   "Area03_Messages".W.Msg[#WngIndex + 0] := "A0301_Fermi_P4".Warning.Fermi[1].NotAutReady;
   "Area03_Messages".W.Msg[#WngIndex + 1] := "A0301_Fermi_P4".Warning.Fermi[1].PressureRunning_Timeout;
   "Area03_Messages".W.Msg[#WngIndex + 2] := "A0301_Fermi_P4".Warning.Fermi[1].Rest_MissingExtEnable;
   "Area03_Messages".W.Msg[#WngIndex + 3] := "A0301_Fermi_P4".Warning.Fermi[1].Work_MissingExtEnable;
   "Area03_Messages".W.Msg[#WngIndex + 4] := "A0301_Fermi_P4".Warning.Fermi[1].Missing_Rest_Ls_ON[1];
   "Area03_Messages".W.Msg[#WngIndex + 5] := "A0301_Fermi_P4".Warning.Fermi[1].Missing_Work_Ls_ON[1];
   "Area03_Messages".W.Msg[#WngIndex + 6] := "A0301_Fermi_P4".Warning.Fermi[2].NotAutReady;
   "Area03_Messages".W.Msg[#WngIndex + 7] := "A0301_Fermi_P4".Warning.Fermi[2].PressureRunning_Timeout;
   "Area03_Messages".W.Msg[#WngIndex + 8] := "A0301_Fermi_P4".Warning.Fermi[2].Rest_MissingExtEnable;
   "Area03_Messages".W.Msg[#WngIndex + 9] := "A0301_Fermi_P4".Warning.Fermi[2].Work_MissingExtEnable;
   "Area03_Messages".W.Msg[#WngIndex + 10] := "A0301_Fermi_P4".Warning.Fermi[2].Missing_Rest_Ls_ON[1];
   "Area03_Messages".W.Msg[#WngIndex + 11] := "A0301_Fermi_P4".Warning.Fermi[2].Missing_Work_Ls_ON[1];
   "Area03_Messages".W.Msg[#WngIndex + 12] := "A0301_Fermi_P4".Warning.Fermi[3].NotAutReady;
   "Area03_Messages".W.Msg[#WngIndex + 13] := "A0301_Fermi_P4".Warning.Fermi[3].PressureRunning_Timeout;
   "Area03_Messages".W.Msg[#WngIndex + 14] := "A0301_Fermi_P4".Warning.Fermi[3].Rest_MissingExtEnable;
   "Area03_Messages".W.Msg[#WngIndex + 15] := "A0301_Fermi_P4".Warning.Fermi[3].Work_MissingExtEnable;
   "Area03_Messages".W.Msg[#WngIndex + 16] := "A0301_Fermi_P4".Warning.Fermi[3].Missing_Rest_Ls_ON[1];
   "Area03_Messages".W.Msg[#WngIndex + 17] := "A0301_Fermi_P4".Warning.Fermi[3].Missing_Work_Ls_ON[1];
   "Area03_Messages".W.Msg[#WngIndex + 18] := "A0301_Fermi_P4".Warning.Fermi[4].NotAutReady;
   "Area03_Messages".W.Msg[#WngIndex + 19] := "A0301_Fermi_P4".Warning.Fermi[4].PressureRunning_Timeout;
   "Area03_Messages".W.Msg[#WngIndex + 20] := "A0301_Fermi_P4".Warning.Fermi[4].Rest_MissingExtEnable;
   "Area03_Messages".W.Msg[#WngIndex + 21] := "A0301_Fermi_P4".Warning.Fermi[4].Work_MissingExtEnable;
   "Area03_Messages".W.Msg[#WngIndex + 22] := "A0301_Fermi_P4".Warning.Fermi[4].Missing_Rest_Ls_ON[1];
   "Area03_Messages".W.Msg[#WngIndex + 23] := "A0301_Fermi_P4".Warning.Fermi[4].Missing_Work_Ls_ON[1];
   "Area03_Messages".W.Msg[#WngIndex + 24] := "A0301_Fermi_P4".Warning.Fermi[5].NotAutReady;
   "Area03_Messages".W.Msg[#WngIndex + 25] := "A0301_Fermi_P4".Warning.Fermi[5].PressureRunning_Timeout;
   "Area03_Messages".W.Msg[#WngIndex + 26] := "A0301_Fermi_P4".Warning.Fermi[5].Rest_MissingExtEnable;
   "Area03_Messages".W.Msg[#WngIndex + 27] := "A0301_Fermi_P4".Warning.Fermi[5].Work_MissingExtEnable;
   "Area03_Messages".W.Msg[#WngIndex + 28] := "A0301_Fermi_P4".Warning.Fermi[5].Missing_Rest_Ls_ON[1];
   "Area03_Messages".W.Msg[#WngIndex + 29] := "A0301_Fermi_P4".Warning.Fermi[5].Missing_Work_Ls_ON[1];
   "Area03_Messages".W.Msg[#WngIndex + 30] := "A0301_Fermi_P4".Warning.Fermi[6].NotAutReady;
   "Area03_Messages".W.Msg[#WngIndex + 31] := "A0301_Fermi_P4".Warning.Fermi[6].PressureRunning_Timeout;
   "Area03_Messages".W.Msg[#WngIndex + 32] := "A0301_Fermi_P4".Warning.Fermi[6].Rest_MissingExtEnable;
   "Area03_Messages".W.Msg[#WngIndex + 33] := "A0301_Fermi_P4".Warning.Fermi[6].Work_MissingExtEnable;
   "Area03_Messages".W.Msg[#WngIndex + 34] := "A0301_Fermi_P4".Warning.Fermi[6].Missing_Rest_Ls_ON[1];
   "Area03_Messages".W.Msg[#WngIndex + 35] := "A0301_Fermi_P4".Warning.Fermi[6].Missing_Work_Ls_ON[1];
   "Area03_Messages".W.Msg[#WngIndex + 36] := FALSE;
   "Area03_Messages".W.Msg[#WngIndex + 37] := FALSE;
   "Area03_Messages".W.Msg[#WngIndex + 38] := "A0301_Fermi_P4".Warning.OP_REST_MissingCnd;
   "Area03_Messages".W.Msg[#WngIndex + 39] := "A0301_Fermi_P4".Warning.OP_WORK_MissingCnd;

   //Spintore Laterale
   // 
   #WngIndex := 330;

   "Area03_Messages".W.Msg[#WngIndex + 0] := "A0301_Spintore_Lat".Warning.Vrt_1.NotAutReady;
   "Area03_Messages".W.Msg[#WngIndex + 1] := "A0301_Spintore_Lat".Warning.Vrt_1.PressureRunning_Timeout;
   "Area03_Messages".W.Msg[#WngIndex + 2] := "A0301_Spintore_Lat".Warning.Vrt_1.Rest_MissingExtEnable;
   "Area03_Messages".W.Msg[#WngIndex + 3] := "A0301_Spintore_Lat".Warning.Vrt_1.Work_MissingExtEnable;
   "Area03_Messages".W.Msg[#WngIndex + 4] := "A0301_Spintore_Lat".Warning.Vrt_1.Missing_Rest_Ls_ON[1];
   "Area03_Messages".W.Msg[#WngIndex + 5] := "A0301_Spintore_Lat".Warning.Vrt_1.Missing_Work_Ls_ON[1];
   "Area03_Messages".W.Msg[#WngIndex + 6] := FALSE;
   "Area03_Messages".W.Msg[#WngIndex + 7] := "A0301_Spintore_Lat".Warning.Orz_1.NotAutReady;;
   "Area03_Messages".W.Msg[#WngIndex + 8] := "A0301_Spintore_Lat".Warning.Orz_1.PressureRunning_Timeout;
   "Area03_Messages".W.Msg[#WngIndex + 9] := "A0301_Spintore_Lat".Warning.Orz_1.Rest_MissingExtEnable;
   "Area03_Messages".W.Msg[#WngIndex + 10] := "A0301_Spintore_Lat".Warning.Orz_1.Work_MissingExtEnable;
   "Area03_Messages".W.Msg[#WngIndex + 11] := "A0301_Spintore_Lat".Warning.Orz_1.Missing_Rest_Ls_ON[1];
   "Area03_Messages".W.Msg[#WngIndex + 12] := "A0301_Spintore_Lat".Warning.Orz_1.Missing_Work_Ls_ON[1];
   "Area03_Messages".W.Msg[#WngIndex + 13] := FALSE;
   "Area03_Messages".W.Msg[#WngIndex + 14] := "A0301_Spintore_Lat".Warning.Orz_1_AnalSens.SensorDisabled;
   "Area03_Messages".W.Msg[#WngIndex + 15] := "A0301_Spintore_Lat".Warning.Orz_1_AnalSens.PresetNeed;;
   "Area03_Messages".W.Msg[#WngIndex + 16] := "A0301_Spintore_Lat".Warning.Orz_1_AnalSens.SignalError;
   "Area03_Messages".W.Msg[#WngIndex + 17] := FALSE;
   "Area03_Messages".W.Msg[#WngIndex + 18] := "A0301_Spintore_Lat".Warning.OP_REST_MissingCnd;
   "Area03_Messages".W.Msg[#WngIndex + 19] := "A0301_Spintore_Lat".Warning.OP_WORK_MissingCnd;
   "Area03_Messages".W.Msg[#WngIndex + 20] := "A0301_Spintore_Lat".Warning.Vrt_2.NotAutReady;;
   "Area03_Messages".W.Msg[#WngIndex + 21] := "A0301_Spintore_Lat".Warning.Vrt_2.PressureRunning_Timeout;
   "Area03_Messages".W.Msg[#WngIndex + 22] := "A0301_Spintore_Lat".Warning.Vrt_2.Rest_MissingExtEnable;
   "Area03_Messages".W.Msg[#WngIndex + 23] := "A0301_Spintore_Lat".Warning.Vrt_2.Work_MissingExtEnable;
   "Area03_Messages".W.Msg[#WngIndex + 24] := "A0301_Spintore_Lat".Warning.Vrt_2.Missing_Rest_Ls_ON[1];
   "Area03_Messages".W.Msg[#WngIndex + 25] := "A0301_Spintore_Lat".Warning.Vrt_2.Missing_Work_Ls_ON[1];
   "Area03_Messages".W.Msg[#WngIndex + 26] := FALSE;
   "Area03_Messages".W.Msg[#WngIndex + 27] := "A0301_Spintore_Lat".Warning.Orz_2.NotAutReady;
   "Area03_Messages".W.Msg[#WngIndex + 28] := "A0301_Spintore_Lat".Warning.Orz_2.PressureRunning_Timeout;
   "Area03_Messages".W.Msg[#WngIndex + 29] := "A0301_Spintore_Lat".Warning.Orz_2.Rest_MissingExtEnable;
   "Area03_Messages".W.Msg[#WngIndex + 30] := "A0301_Spintore_Lat".Warning.Orz_2.Work_MissingExtEnable;
   "Area03_Messages".W.Msg[#WngIndex + 31] := "A0301_Spintore_Lat".Warning.Orz_2.Missing_Rest_Ls_ON[1];
   "Area03_Messages".W.Msg[#WngIndex + 32] := "A0301_Spintore_Lat".Warning.Orz_2.Missing_Work_Ls_ON[1];
   "Area03_Messages".W.Msg[#WngIndex + 33] := "A0301_Spintore_Lat".Warning.Orz_2_AnalSens.SensorDisabled;
   "Area03_Messages".W.Msg[#WngIndex + 34] := "A0301_Spintore_Lat".Warning.Orz_2_AnalSens.PresetNeed;
   "Area03_Messages".W.Msg[#WngIndex + 35] := "A0301_Spintore_Lat".Warning.Orz_2_AnalSens.SignalError;
   "Area03_Messages".W.Msg[#WngIndex + 36] := "A0301_Spintore_Lat".Warning.Finestre.SpinLat1_SpinLong_Stop;
   "Area03_Messages".W.Msg[#WngIndex + 37] := "A0301_Spintore_Lat".Warning.Finestre.SpinLat2_SpinLong_Stop;


   //Spintore Longitudinale
   // 
   #WngIndex := 380;

   "Area03_Messages".W.Msg[#WngIndex + 0] := "A0301_Spintore_Lat".Warning.Sollevatori[1].NotAutReady;
   "Area03_Messages".W.Msg[#WngIndex + 1] := "A0301_Spintore_Lat".Warning.Sollevatori[1].PressureRunning_Timeout;
   "Area03_Messages".W.Msg[#WngIndex + 2] := "A0301_Spintore_Lat".Warning.Sollevatori[1].Rest_MissingExtEnable;
   "Area03_Messages".W.Msg[#WngIndex + 3] := "A0301_Spintore_Lat".Warning.Sollevatori[1].Work_MissingExtEnable;
   "Area03_Messages".W.Msg[#WngIndex + 4] := "A0301_Spintore_Lat".Warning.Sollevatori[1].Missing_Rest_Ls_ON[1];
   "Area03_Messages".W.Msg[#WngIndex + 5] := "A0301_Spintore_Lat".Warning.Sollevatori[1].Missing_Work_Ls_ON[1];
   "Area03_Messages".W.Msg[#WngIndex + 6] := FALSE;
   "Area03_Messages".W.Msg[#WngIndex + 7] := "A0301_Spintore_Lat".Warning.Sollevatori[2].NotAutReady;;
   "Area03_Messages".W.Msg[#WngIndex + 8] := "A0301_Spintore_Lat".Warning.Sollevatori[2].PressureRunning_Timeout;
   "Area03_Messages".W.Msg[#WngIndex + 9] := "A0301_Spintore_Lat".Warning.Sollevatori[2].Rest_MissingExtEnable;
   "Area03_Messages".W.Msg[#WngIndex + 10] := "A0301_Spintore_Lat".Warning.Sollevatori[2].Work_MissingExtEnable;
   "Area03_Messages".W.Msg[#WngIndex + 11] := "A0301_Spintore_Lat".Warning.Sollevatori[2].Missing_Rest_Ls_ON[1];
   "Area03_Messages".W.Msg[#WngIndex + 12] := "A0301_Spintore_Lat".Warning.Sollevatori[2].Missing_Work_Ls_ON[1];
   "Area03_Messages".W.Msg[#WngIndex + 13] := FALSE;
   "Area03_Messages".W.Msg[#WngIndex + 14] := "A0301_Spintore_Lat".Warning.Sollevatori[3].NotAutReady;
   "Area03_Messages".W.Msg[#WngIndex + 15] := "A0301_Spintore_Lat".Warning.Sollevatori[3].PressureRunning_Timeout;
   "Area03_Messages".W.Msg[#WngIndex + 16] := "A0301_Spintore_Lat".Warning.Sollevatori[3].Rest_MissingExtEnable;
   "Area03_Messages".W.Msg[#WngIndex + 17] := "A0301_Spintore_Lat".Warning.Sollevatori[3].Work_MissingExtEnable;
   "Area03_Messages".W.Msg[#WngIndex + 18] := "A0301_Spintore_Lat".Warning.Sollevatori[3].Missing_Rest_Ls_ON[1];
   "Area03_Messages".W.Msg[#WngIndex + 19] := "A0301_Spintore_Lat".Warning.Sollevatori[3].Missing_Work_Ls_ON[1];
   "Area03_Messages".W.Msg[#WngIndex + 20] := FALSE;
   "Area03_Messages".W.Msg[#WngIndex + 21] := "A0301_Spintore_Lat".Warning.Sollevatori[4].NotAutReady;
   "Area03_Messages".W.Msg[#WngIndex + 22] := "A0301_Spintore_Lat".Warning.Sollevatori[4].PressureRunning_Timeout;
   "Area03_Messages".W.Msg[#WngIndex + 23] := "A0301_Spintore_Lat".Warning.Sollevatori[4].Rest_MissingExtEnable;
   "Area03_Messages".W.Msg[#WngIndex + 24] := "A0301_Spintore_Lat".Warning.Sollevatori[4].Work_MissingExtEnable;
   "Area03_Messages".W.Msg[#WngIndex + 25] := "A0301_Spintore_Lat".Warning.Sollevatori[4].Missing_Rest_Ls_ON[1];
   "Area03_Messages".W.Msg[#WngIndex + 26] := "A0301_Spintore_Lat".Warning.Sollevatori[4].Missing_Work_Ls_ON[1];
   "Area03_Messages".W.Msg[#WngIndex + 27] := FALSE;
   "Area03_Messages".W.Msg[#WngIndex + 28] := "A0301_Spintore_Lat".Warning.Sollevatori[5].NotAutReady;
   "Area03_Messages".W.Msg[#WngIndex + 29] := "A0301_Spintore_Lat".Warning.Sollevatori[5].PressureRunning_Timeout;
   "Area03_Messages".W.Msg[#WngIndex + 30] := "A0301_Spintore_Lat".Warning.Sollevatori[5].Rest_MissingExtEnable;
   "Area03_Messages".W.Msg[#WngIndex + 31] := "A0301_Spintore_Lat".Warning.Sollevatori[5].Work_MissingExtEnable;
   "Area03_Messages".W.Msg[#WngIndex + 32] := "A0301_Spintore_Lat".Warning.Sollevatori[5].Missing_Rest_Ls_ON[1];
   "Area03_Messages".W.Msg[#WngIndex + 33] := "A0301_Spintore_Lat".Warning.Sollevatori[5].Missing_Work_Ls_ON[1];
   "Area03_Messages".W.Msg[#WngIndex + 34] := FALSE;
   "Area03_Messages".W.Msg[#WngIndex + 35] := "A0301_Spintore_Lat".Warning.Sollevatori[6].NotAutReady;
   "Area03_Messages".W.Msg[#WngIndex + 36] := "A0301_Spintore_Lat".Warning.Sollevatori[6].PressureRunning_Timeout;
   "Area03_Messages".W.Msg[#WngIndex + 37] := "A0301_Spintore_Lat".Warning.Sollevatori[6].Rest_MissingExtEnable;
   "Area03_Messages".W.Msg[#WngIndex + 38] := "A0301_Spintore_Lat".Warning.Sollevatori[6].Work_MissingExtEnable;
   "Area03_Messages".W.Msg[#WngIndex + 39] := "A0301_Spintore_Lat".Warning.Sollevatori[6].Missing_Rest_Ls_ON[1];
   "Area03_Messages".W.Msg[#WngIndex + 40] := "A0301_Spintore_Lat".Warning.Sollevatori[6].Missing_Work_Ls_ON[1];
   "Area03_Messages".W.Msg[#WngIndex + 41] := FALSE;
   "Area03_Messages".W.Msg[#WngIndex + 42] := "A0301_Spintore_Lat".Warning.Sollevatori[7].NotAutReady;
   "Area03_Messages".W.Msg[#WngIndex + 43] := "A0301_Spintore_Lat".Warning.Sollevatori[7].PressureRunning_Timeout;
   "Area03_Messages".W.Msg[#WngIndex + 44] := "A0301_Spintore_Lat".Warning.Sollevatori[7].Rest_MissingExtEnable;
   "Area03_Messages".W.Msg[#WngIndex + 45] := "A0301_Spintore_Lat".Warning.Sollevatori[7].Work_MissingExtEnable;
   "Area03_Messages".W.Msg[#WngIndex + 46] := "A0301_Spintore_Lat".Warning.Sollevatori[7].Missing_Rest_Ls_ON[1];
   "Area03_Messages".W.Msg[#WngIndex + 47] := "A0301_Spintore_Lat".Warning.Sollevatori[7].Missing_Work_Ls_ON[1];
   "Area03_Messages".W.Msg[#WngIndex + 48] := FALSE;
   "Area03_Messages".W.Msg[#WngIndex + 49] := FALSE;



   //Manager stazioni pareggiamento
   // 
   #WngIndex := 430;

   "Area03_Messages".W.Msg[#WngIndex + 0] := "A0302_Manager".Warning.CheckBancoAccumulo;
   "Area03_Messages".W.Msg[#WngIndex + 1] := FALSE;
   "Area03_Messages".W.Msg[#WngIndex + 2] := FALSE;
   "Area03_Messages".W.Msg[#WngIndex + 3] := FALSE;
   "Area03_Messages".W.Msg[#WngIndex + 4] := FALSE;
   "Area03_Messages".W.Msg[#WngIndex + 5] := FALSE;
   "Area03_Messages".W.Msg[#WngIndex + 6] := FALSE;
   "Area03_Messages".W.Msg[#WngIndex + 7] := FALSE;
   "Area03_Messages".W.Msg[#WngIndex + 8] := FALSE;
   "Area03_Messages".W.Msg[#WngIndex + 9] := FALSE;

   //HU CYTROPACK
   // 
   #WngIndex := 440;

   "Area03_Messages".W.Msg[#WngIndex + 0] := FALSE;
   "Area03_Messages".W.Msg[#WngIndex + 1] := FALSE;
   "Area03_Messages".W.Msg[#WngIndex + 2] := FALSE;
   "Area03_Messages".W.Msg[#WngIndex + 3] := FALSE;
   "Area03_Messages".W.Msg[#WngIndex + 4] := FALSE;
   "Area03_Messages".W.Msg[#WngIndex + 5] := FALSE;
   "Area03_Messages".W.Msg[#WngIndex + 6] := FALSE;
   "Area03_Messages".W.Msg[#WngIndex + 7] := FALSE;
   "Area03_Messages".W.Msg[#WngIndex + 8] := FALSE;
   "Area03_Messages".W.Msg[#WngIndex + 9] := FALSE;
   "Area03_Messages".W.Msg[#WngIndex + 10] := FALSE;
   "Area03_Messages".W.Msg[#WngIndex + 11] := FALSE;
   "Area03_Messages".W.Msg[#WngIndex + 12] := FALSE;
   "Area03_Messages".W.Msg[#WngIndex + 13] := FALSE;
   "Area03_Messages".W.Msg[#WngIndex + 14] := FALSE;
   "Area03_Messages".W.Msg[#WngIndex + 15] := FALSE;
   "Area03_Messages".W.Msg[#WngIndex + 16] := FALSE;
   "Area03_Messages".W.Msg[#WngIndex + 17] := FALSE;
   "Area03_Messages".W.Msg[#WngIndex + 18] := FALSE;
   "Area03_Messages".W.Msg[#WngIndex + 19] := FALSE;

   //Spintore
   // 
   #WngIndex := 470;

   "Area03_Messages".W.Msg[#WngIndex + 0] := "A0302_Spintore".Warning.Ax.NotAutReady;
   "Area03_Messages".W.Msg[#WngIndex + 1] := "A0302_Spintore".Warning.Ax.Minus_CndMissing;
   "Area03_Messages".W.Msg[#WngIndex + 2] := "A0302_Spintore".Warning.Ax.Plus_CndMissing;
   "Area03_Messages".W.Msg[#WngIndex + 3] := "A0302_Spintore".Warning.Ax.S120_Warning;
   "Area03_Messages".W.Msg[#WngIndex + 4] := "A0302_Spintore".Warning.Ax.Ax_NotHomed;
   "Area03_Messages".W.Msg[#WngIndex + 5] := "A0302_Spintore".Warning.Ax.Ax_FlyingHome;
   "Area03_Messages".W.Msg[#WngIndex + 6] := "A0302_Spintore".Warning.Ax.Ax_SwLimitMinus;
   "Area03_Messages".W.Msg[#WngIndex + 7] := "A0302_Spintore".Warning.Ax.Ax_SwLimitPlus;
   "Area03_Messages".W.Msg[#WngIndex + 8] := FALSE;
   "Area03_Messages".W.Msg[#WngIndex + 9] := FALSE;
   "Area03_Messages".W.Msg[#WngIndex + 10] := "A0302_Spintore".Warning.Vrt.NotAutReady;
   "Area03_Messages".W.Msg[#WngIndex + 11] := "A0302_Spintore".Warning.Vrt.PressureRunning_Timeout;
   "Area03_Messages".W.Msg[#WngIndex + 12] := "A0302_Spintore".Warning.Vrt.Rest_MissingExtEnable;
   "Area03_Messages".W.Msg[#WngIndex + 13] := "A0302_Spintore".Warning.Vrt.Work_MissingExtEnable;
   "Area03_Messages".W.Msg[#WngIndex + 14] := "A0302_Spintore".Warning.Vrt.Missing_Rest_Ls_ON[1];
   "Area03_Messages".W.Msg[#WngIndex + 15] := "A0302_Spintore".Warning.Vrt.Missing_Work_Ls_ON[1];
   "Area03_Messages".W.Msg[#WngIndex + 16] := FALSE;
   "Area03_Messages".W.Msg[#WngIndex + 17] := FALSE;
   "Area03_Messages".W.Msg[#WngIndex + 18] := "A0302_Spintore".Warning.Orz.NotAutReady;
   "Area03_Messages".W.Msg[#WngIndex + 19] := "A0302_Spintore".Warning.Orz.PressureRunning_Timeout;
   "Area03_Messages".W.Msg[#WngIndex + 20] := "A0302_Spintore".Warning.Orz.Rest_MissingExtEnable;
   "Area03_Messages".W.Msg[#WngIndex + 21] := "A0302_Spintore".Warning.Orz.Work_MissingExtEnable;
   "Area03_Messages".W.Msg[#WngIndex + 22] := "A0302_Spintore".Warning.Orz.Missing_Rest_Ls_ON[1];
   "Area03_Messages".W.Msg[#WngIndex + 23] := "A0302_Spintore".Warning.Orz.Missing_Work_Ls_ON[1];
   "Area03_Messages".W.Msg[#WngIndex + 24] := FALSE;
   "Area03_Messages".W.Msg[#WngIndex + 25] := FALSE;
   "Area03_Messages".W.Msg[#WngIndex + 26] := "A0302_Spintore".Warning.Orz_AnalSens.SensorDisabled;
   "Area03_Messages".W.Msg[#WngIndex + 27] := "A0302_Spintore".Warning.Orz_AnalSens.PresetNeed;
   "Area03_Messages".W.Msg[#WngIndex + 28] := "A0302_Spintore".Warning.Orz_AnalSens.SignalError;
   "Area03_Messages".W.Msg[#WngIndex + 29] := FALSE;
   "Area03_Messages".W.Msg[#WngIndex + 30] := FALSE;
   "Area03_Messages".W.Msg[#WngIndex + 31] := "A0302_Spintore".Warning.OP_REST_MissingCnd;
   "Area03_Messages".W.Msg[#WngIndex + 32] := "A0302_Spintore".Warning.OP_WORK_MissingCnd;

   //Bordatrice
   // 
   #WngIndex := 510;

   "Area03_Messages".W.Msg[#WngIndex + 0] := "A0302_Bordatrice".Warning.Ax.NotAutReady;
   "Area03_Messages".W.Msg[#WngIndex + 1] := "A0302_Bordatrice".Warning.Ax.Minus_CndMissing;
   "Area03_Messages".W.Msg[#WngIndex + 2] := "A0302_Bordatrice".Warning.Ax.Plus_CndMissing;
   "Area03_Messages".W.Msg[#WngIndex + 3] := "A0302_Bordatrice".Warning.Ax.S120_Warning;
   "Area03_Messages".W.Msg[#WngIndex + 4] := "A0302_Bordatrice".Warning.Ax.Ax_NotHomed;
   "Area03_Messages".W.Msg[#WngIndex + 5] := "A0302_Bordatrice".Warning.Ax.Ax_FlyingHome;
   "Area03_Messages".W.Msg[#WngIndex + 6] := "A0302_Bordatrice".Warning.Ax.Ax_SwLimitMinus;
   "Area03_Messages".W.Msg[#WngIndex + 7] := "A0302_Bordatrice".Warning.Ax.Ax_SwLimitPlus;
   "Area03_Messages".W.Msg[#WngIndex + 8] := "A0302_Bordatrice".Warning.OP_REST_MissingCnd;
   "Area03_Messages".W.Msg[#WngIndex + 9] := "A0302_Bordatrice".Warning.OP_WORK_MissingCnd;
   "Area03_Messages".W.Msg[#WngIndex + 10] := FALSE;
   "Area03_Messages".W.Msg[#WngIndex + 11] := FALSE;
   "Area03_Messages".W.Msg[#WngIndex + 12] := FALSE;
   "Area03_Messages".W.Msg[#WngIndex + 13] := FALSE;
   "Area03_Messages".W.Msg[#WngIndex + 14] := FALSE;
   "Area03_Messages".W.Msg[#WngIndex + 15] := FALSE;
   "Area03_Messages".W.Msg[#WngIndex + 16] := FALSE;
   "Area03_Messages".W.Msg[#WngIndex + 17] := FALSE;
   "Area03_Messages".W.Msg[#WngIndex + 18] := FALSE;
   "Area03_Messages".W.Msg[#WngIndex + 19] := FALSE;
   "Area03_Messages".W.Msg[#WngIndex + 20] := FALSE;


   //Rulliera
   // 
   #WngIndex := 540;

   "Area03_Messages".W.Msg[#WngIndex + 0] := "A0302_Rulliera".Warning.Rulliera[1].NotAutReady;
   "Area03_Messages".W.Msg[#WngIndex + 1] := "A0302_Rulliera".Warning.Rulliera[1].MissingCnd_Bkw;
   "Area03_Messages".W.Msg[#WngIndex + 2] := "A0302_Rulliera".Warning.Rulliera[1].MissingCnd_Fwd;
   "Area03_Messages".W.Msg[#WngIndex + 3] := "A0302_Rulliera".Warning.Rulliera[1].Ax.Drive;
   "Area03_Messages".W.Msg[#WngIndex + 4] := "A0302_Rulliera".Warning.Rulliera[2].NotAutReady;
   "Area03_Messages".W.Msg[#WngIndex + 5] := "A0302_Rulliera".Warning.Rulliera[2].MissingCnd_Bkw;
   "Area03_Messages".W.Msg[#WngIndex + 6] := "A0302_Rulliera".Warning.Rulliera[2].MissingCnd_Fwd;
   "Area03_Messages".W.Msg[#WngIndex + 7] := "A0302_Rulliera".Warning.Rulliera[2].Ax.Drive;
   "Area03_Messages".W.Msg[#WngIndex + 8] := "A0302_Rulliera".Warning.OP_REST_MissingCnd;
   "Area03_Messages".W.Msg[#WngIndex + 9] := "A0302_Rulliera".Warning.OP_WORK_MissingCnd;
   "Area03_Messages".W.Msg[#WngIndex + 10] := FALSE;
   "Area03_Messages".W.Msg[#WngIndex + 11] := FALSE;
   "Area03_Messages".W.Msg[#WngIndex + 12] := FALSE;
   "Area03_Messages".W.Msg[#WngIndex + 13] := FALSE;
   "Area03_Messages".W.Msg[#WngIndex + 14] := FALSE;
   "Area03_Messages".W.Msg[#WngIndex + 15] := FALSE;
   "Area03_Messages".W.Msg[#WngIndex + 16] := FALSE;
   "Area03_Messages".W.Msg[#WngIndex + 17] := FALSE;
   "Area03_Messages".W.Msg[#WngIndex + 18] := FALSE;
   "Area03_Messages".W.Msg[#WngIndex + 19] := FALSE;


   //Centratori
   // 
   #WngIndex := 560;

   "Area03_Messages".W.Msg[#WngIndex + 0] := "A0302_Centratori".Warning.Centratore[1].NotAutReady;
   "Area03_Messages".W.Msg[#WngIndex + 1] := "A0302_Centratori".Warning.Centratore[1].PressureRunning_Timeout;
   "Area03_Messages".W.Msg[#WngIndex + 2] := "A0302_Centratori".Warning.Centratore[1].Rest_MissingExtEnable;
   "Area03_Messages".W.Msg[#WngIndex + 3] := "A0302_Centratori".Warning.Centratore[1].Work_MissingExtEnable;
   "Area03_Messages".W.Msg[#WngIndex + 4] := "A0302_Centratori".Warning.Centratore[1].Missing_Rest_Ls_ON[1];
   "Area03_Messages".W.Msg[#WngIndex + 5] := "A0302_Centratori".Warning.Centratore[1].Missing_Work_Ls_ON[1];
   "Area03_Messages".W.Msg[#WngIndex + 6] := FALSE;
   "Area03_Messages".W.Msg[#WngIndex + 7] := FALSE;
   "Area03_Messages".W.Msg[#WngIndex + 8] := "A0302_Centratori".Warning.Centratore[2].NotAutReady;
   "Area03_Messages".W.Msg[#WngIndex + 9] := "A0302_Centratori".Warning.Centratore[2].PressureRunning_Timeout;
   "Area03_Messages".W.Msg[#WngIndex + 10] := "A0302_Centratori".Warning.Centratore[2].Rest_MissingExtEnable;
   "Area03_Messages".W.Msg[#WngIndex + 11] := "A0302_Centratori".Warning.Centratore[2].Work_MissingExtEnable;
   "Area03_Messages".W.Msg[#WngIndex + 12] := "A0302_Centratori".Warning.Centratore[2].Missing_Rest_Ls_ON[1];
   "Area03_Messages".W.Msg[#WngIndex + 13] := "A0302_Centratori".Warning.Centratore[2].Missing_Work_Ls_ON[1];
   "Area03_Messages".W.Msg[#WngIndex + 14] := FALSE;
   "Area03_Messages".W.Msg[#WngIndex + 15] := FALSE;
   "Area03_Messages".W.Msg[#WngIndex + 16] := "A0302_Centratori".Warning.Centratore[3].NotAutReady;
   "Area03_Messages".W.Msg[#WngIndex + 17] := "A0302_Centratori".Warning.Centratore[3].PressureRunning_Timeout;
   "Area03_Messages".W.Msg[#WngIndex + 18] := "A0302_Centratori".Warning.Centratore[3].Rest_MissingExtEnable;
   "Area03_Messages".W.Msg[#WngIndex + 19] := "A0302_Centratori".Warning.Centratore[3].Work_MissingExtEnable;
   "Area03_Messages".W.Msg[#WngIndex + 20] := "A0302_Centratori".Warning.Centratore[3].Missing_Rest_Ls_ON[1];
   "Area03_Messages".W.Msg[#WngIndex + 21] := "A0302_Centratori".Warning.Centratore[3].Missing_Work_Ls_ON[1];
   "Area03_Messages".W.Msg[#WngIndex + 22] := FALSE;
   "Area03_Messages".W.Msg[#WngIndex + 23] := FALSE;
   "Area03_Messages".W.Msg[#WngIndex + 24] := "A0302_Centratori".Warning.Sollevamento[1].NotAutReady;
   "Area03_Messages".W.Msg[#WngIndex + 25] := "A0302_Centratori".Warning.Sollevamento[1].PressureRunning_Timeout;
   "Area03_Messages".W.Msg[#WngIndex + 26] := "A0302_Centratori".Warning.Sollevamento[1].Rest_MissingExtEnable;
   "Area03_Messages".W.Msg[#WngIndex + 27] := "A0302_Centratori".Warning.Sollevamento[1].Work_MissingExtEnable;
   "Area03_Messages".W.Msg[#WngIndex + 28] := "A0302_Centratori".Warning.Sollevamento[1].Missing_Rest_Ls_ON[1];
   "Area03_Messages".W.Msg[#WngIndex + 29] := "A0302_Centratori".Warning.Sollevamento[1].Missing_Work_Ls_ON[1];
   "Area03_Messages".W.Msg[#WngIndex + 30] := FALSE;
   "Area03_Messages".W.Msg[#WngIndex + 31] := FALSE;
   "Area03_Messages".W.Msg[#WngIndex + 32] := "A0302_Centratori".Warning.Sollevamento[2].NotAutReady;
   "Area03_Messages".W.Msg[#WngIndex + 33] := "A0302_Centratori".Warning.Sollevamento[2].PressureRunning_Timeout;
   "Area03_Messages".W.Msg[#WngIndex + 34] := "A0302_Centratori".Warning.Sollevamento[2].Rest_MissingExtEnable;
   "Area03_Messages".W.Msg[#WngIndex + 35] := "A0302_Centratori".Warning.Sollevamento[2].Work_MissingExtEnable;
   "Area03_Messages".W.Msg[#WngIndex + 36] := "A0302_Centratori".Warning.Sollevamento[2].Missing_Rest_Ls_ON[1];
   "Area03_Messages".W.Msg[#WngIndex + 37] := "A0302_Centratori".Warning.Sollevamento[2].Missing_Work_Ls_ON[1];
   "Area03_Messages".W.Msg[#WngIndex + 38] := FALSE;
   "Area03_Messages".W.Msg[#WngIndex + 39] := FALSE;
   "Area03_Messages".W.Msg[#WngIndex + 40] := "A0302_Centratori".Warning.Sollevamento[3].NotAutReady;
   "Area03_Messages".W.Msg[#WngIndex + 41] := "A0302_Centratori".Warning.Sollevamento[3].PressureRunning_Timeout;
   "Area03_Messages".W.Msg[#WngIndex + 42] := "A0302_Centratori".Warning.Sollevamento[3].Rest_MissingExtEnable;
   "Area03_Messages".W.Msg[#WngIndex + 43] := "A0302_Centratori".Warning.Sollevamento[3].Work_MissingExtEnable;
   "Area03_Messages".W.Msg[#WngIndex + 44] := "A0302_Centratori".Warning.Sollevamento[3].Missing_Rest_Ls_ON[1];
   "Area03_Messages".W.Msg[#WngIndex + 45] := "A0302_Centratori".Warning.Sollevamento[3].Missing_Work_Ls_ON[1];
   "Area03_Messages".W.Msg[#WngIndex + 46] := FALSE;
   "Area03_Messages".W.Msg[#WngIndex + 47] := FALSE;
   "Area03_Messages".W.Msg[#WngIndex + 48] := "A0302_Centratori".Warning.OP_REST_Centr_MissingCnd;
   "Area03_Messages".W.Msg[#WngIndex + 49] := "A0302_Centratori".Warning.OP_WORK_Centr_MissingCnd;

   //Pareggiatore Coda
   // 
   #WngIndex := 610;

   "Area03_Messages".W.Msg[#WngIndex + 0] := "A0302_PareggiatoreCoda".Warning.Ax.NotAutReady;
   "Area03_Messages".W.Msg[#WngIndex + 1] := "A0302_PareggiatoreCoda".Warning.Ax.MissingCnd_Minus;
   "Area03_Messages".W.Msg[#WngIndex + 2] := "A0302_PareggiatoreCoda".Warning.Ax.MissingCnd_Plus;
   "Area03_Messages".W.Msg[#WngIndex + 3] := "A0302_PareggiatoreCoda".Warning.Ax.Ax_NotHomed;
   "Area03_Messages".W.Msg[#WngIndex + 4] := "A0302_PareggiatoreCoda".Warning.Ax.Ax.SwLimitMinus;
   "Area03_Messages".W.Msg[#WngIndex + 5] := "A0302_PareggiatoreCoda".Warning.Ax.Ax.SwLimitPlus;
   "Area03_Messages".W.Msg[#WngIndex + 6] := "A0302_PareggiatoreCoda".Warning.Ax.S120.Drive;
   "Area03_Messages".W.Msg[#WngIndex + 7] := FALSE;
   "Area03_Messages".W.Msg[#WngIndex + 8] := FALSE;
   "Area03_Messages".W.Msg[#WngIndex + 9] := FALSE;
   "Area03_Messages".W.Msg[#WngIndex + 10] := "A0302_PareggiatoreCoda".Warning.Bloccaggio.NotAutReady;
   "Area03_Messages".W.Msg[#WngIndex + 11] := "A0302_PareggiatoreCoda".Warning.Bloccaggio.PressureRunning_Timeout;
   "Area03_Messages".W.Msg[#WngIndex + 12] := "A0302_PareggiatoreCoda".Warning.Bloccaggio.Rest_MissingExtEnable;
   "Area03_Messages".W.Msg[#WngIndex + 13] := "A0302_PareggiatoreCoda".Warning.Bloccaggio.Work_MissingExtEnable;
   "Area03_Messages".W.Msg[#WngIndex + 14] := "A0302_PareggiatoreCoda".Warning.Bloccaggio.Missing_Rest_Ls_ON[1];
   "Area03_Messages".W.Msg[#WngIndex + 15] := "A0302_PareggiatoreCoda".Warning.Bloccaggio.Missing_Work_Ls_ON[1];
   "Area03_Messages".W.Msg[#WngIndex + 16] := FALSE;
   "Area03_Messages".W.Msg[#WngIndex + 17] := FALSE;
   "Area03_Messages".W.Msg[#WngIndex + 18] := "A0302_PareggiatoreCoda".Warning.BattutaVerticale.NotAutReady;
   "Area03_Messages".W.Msg[#WngIndex + 19] := "A0302_PareggiatoreCoda".Warning.BattutaVerticale.PressureRunning_Timeout;
   "Area03_Messages".W.Msg[#WngIndex + 20] := "A0302_PareggiatoreCoda".Warning.BattutaVerticale.Rest_MissingExtEnable;
   "Area03_Messages".W.Msg[#WngIndex + 21] := "A0302_PareggiatoreCoda".Warning.BattutaVerticale.Work_MissingExtEnable;
   "Area03_Messages".W.Msg[#WngIndex + 22] := "A0302_PareggiatoreCoda".Warning.BattutaVerticale.Missing_Rest_Ls_ON[1];
   "Area03_Messages".W.Msg[#WngIndex + 23] := "A0302_PareggiatoreCoda".Warning.BattutaVerticale.Missing_Work_Ls_ON[1];
   "Area03_Messages".W.Msg[#WngIndex + 24] := FALSE;
   "Area03_Messages".W.Msg[#WngIndex + 25] := FALSE;
   "Area03_Messages".W.Msg[#WngIndex + 26] := "A0302_PareggiatoreCoda".Warning.PareggiatoreLongitudinale.NotAutReady;
   "Area03_Messages".W.Msg[#WngIndex + 27] := "A0302_PareggiatoreCoda".Warning.PareggiatoreLongitudinale.PressureRunning_Timeout;
   "Area03_Messages".W.Msg[#WngIndex + 28] := "A0302_PareggiatoreCoda".Warning.PareggiatoreLongitudinale.Rest_MissingExtEnable;
   "Area03_Messages".W.Msg[#WngIndex + 29] := "A0302_PareggiatoreCoda".Warning.PareggiatoreLongitudinale.Work_MissingExtEnable;
   "Area03_Messages".W.Msg[#WngIndex + 30] := "A0302_PareggiatoreCoda".Warning.PareggiatoreLongitudinale.Missing_Rest_Ls_ON[1];
   "Area03_Messages".W.Msg[#WngIndex + 31] := "A0302_PareggiatoreCoda".Warning.PareggiatoreLongitudinale.Missing_Work_Ls_ON[1];
   "Area03_Messages".W.Msg[#WngIndex + 32] := FALSE;
   "Area03_Messages".W.Msg[#WngIndex + 33] := FALSE;
   "Area03_Messages".W.Msg[#WngIndex + 34] := "A0302_PareggiatoreCoda".Warning.PosPareggiatoreLong.SensorDisabled;
   "Area03_Messages".W.Msg[#WngIndex + 35] := "A0302_PareggiatoreCoda".Warning.PosPareggiatoreLong.PresetNeed;
   "Area03_Messages".W.Msg[#WngIndex + 36] := "A0302_PareggiatoreCoda".Warning.PosPareggiatoreLong.SignalError;
   "Area03_Messages".W.Msg[#WngIndex + 37] := FALSE;
   "Area03_Messages".W.Msg[#WngIndex + 38] := "A0302_PareggiatoreCoda".Warning.SW_Limit_AntiCollision;
   "Area03_Messages".W.Msg[#WngIndex + 39] := "A0302_PareggiatoreCoda".Warning.MissingCnd.OP_REST_Bloccaggio;
   "Area03_Messages".W.Msg[#WngIndex + 40] := "A0302_PareggiatoreCoda".Warning.MissingCnd.OP_WORK_Bloccaggio;
   "Area03_Messages".W.Msg[#WngIndex + 41] := "A0302_PareggiatoreCoda".Warning.MissingCnd.OP_REST_BattutaVrt;
   "Area03_Messages".W.Msg[#WngIndex + 42] := "A0302_PareggiatoreCoda".Warning.MissingCnd.OP_WORK_BattutaVrt;
   "Area03_Messages".W.Msg[#WngIndex + 43] := "A0302_PareggiatoreCoda".Warning.MissingCnd.OP_REST_PareggLong;
   "Area03_Messages".W.Msg[#WngIndex + 44] := "A0302_PareggiatoreCoda".Warning.MissingCnd.OP_WORK_PareggLong;


   //Pareggiatore Testa
   // 
   #WngIndex := 660;

   "Area03_Messages".W.Msg[#WngIndex + 0] := "A0302_PareggiatoreTesta".Warning.Ax.NotAutReady;
   "Area03_Messages".W.Msg[#WngIndex + 1] := "A0302_PareggiatoreTesta".Warning.Ax.MissingCnd_Minus;
   "Area03_Messages".W.Msg[#WngIndex + 2] := "A0302_PareggiatoreTesta".Warning.Ax.MissingCnd_Plus;
   "Area03_Messages".W.Msg[#WngIndex + 3] := "A0302_PareggiatoreTesta".Warning.Ax.Ax_NotHomed;
   "Area03_Messages".W.Msg[#WngIndex + 4] := "A0302_PareggiatoreTesta".Warning.Ax.Ax.SwLimitMinus;
   "Area03_Messages".W.Msg[#WngIndex + 5] := "A0302_PareggiatoreTesta".Warning.Ax.Ax.SwLimitPlus;
   "Area03_Messages".W.Msg[#WngIndex + 6] := "A0302_PareggiatoreTesta".Warning.Ax.S120.Drive;
   "Area03_Messages".W.Msg[#WngIndex + 7] := FALSE;
   "Area03_Messages".W.Msg[#WngIndex + 8] := FALSE;
   "Area03_Messages".W.Msg[#WngIndex + 9] := FALSE;
   "Area03_Messages".W.Msg[#WngIndex + 10] := "A0302_PareggiatoreTesta".Warning.Bloccaggio.NotAutReady;
   "Area03_Messages".W.Msg[#WngIndex + 11] := "A0302_PareggiatoreTesta".Warning.Bloccaggio.PressureRunning_Timeout;
   "Area03_Messages".W.Msg[#WngIndex + 12] := "A0302_PareggiatoreTesta".Warning.Bloccaggio.Rest_MissingExtEnable;
   "Area03_Messages".W.Msg[#WngIndex + 13] := "A0302_PareggiatoreTesta".Warning.Bloccaggio.Work_MissingExtEnable;
   "Area03_Messages".W.Msg[#WngIndex + 14] := "A0302_PareggiatoreTesta".Warning.Bloccaggio.Missing_Rest_Ls_ON[1];
   "Area03_Messages".W.Msg[#WngIndex + 15] := "A0302_PareggiatoreTesta".Warning.Bloccaggio.Missing_Rest_Ls_ON[2];
   "Area03_Messages".W.Msg[#WngIndex + 16] := "A0302_PareggiatoreTesta".Warning.Bloccaggio.Missing_Work_Ls_ON[1];
   "Area03_Messages".W.Msg[#WngIndex + 17] := "A0302_PareggiatoreTesta".Warning.Bloccaggio.Missing_Work_Ls_ON[2];
   "Area03_Messages".W.Msg[#WngIndex + 18] := "A0302_PareggiatoreTesta".Warning.Sollevamento.NotAutReady;
   "Area03_Messages".W.Msg[#WngIndex + 19] := "A0302_PareggiatoreTesta".Warning.Sollevamento.PressureRunning_Timeout;
   "Area03_Messages".W.Msg[#WngIndex + 20] := "A0302_PareggiatoreTesta".Warning.Sollevamento.Rest_MissingExtEnable;
   "Area03_Messages".W.Msg[#WngIndex + 21] := "A0302_PareggiatoreTesta".Warning.Sollevamento.Work_MissingExtEnable;
   "Area03_Messages".W.Msg[#WngIndex + 22] := "A0302_PareggiatoreTesta".Warning.Sollevamento.Missing_Rest_Ls_ON[1];
   "Area03_Messages".W.Msg[#WngIndex + 23] := "A0302_PareggiatoreTesta".Warning.Sollevamento.Missing_Work_Ls_ON[1];
   "Area03_Messages".W.Msg[#WngIndex + 24] := FALSE;
   "Area03_Messages".W.Msg[#WngIndex + 25] := FALSE;
   "Area03_Messages".W.Msg[#WngIndex + 26] := "A0302_PareggiatoreTesta".Warning.Centraggio.NotAutReady;
   "Area03_Messages".W.Msg[#WngIndex + 27] := "A0302_PareggiatoreTesta".Warning.Centraggio.PressureRunning_Timeout;
   "Area03_Messages".W.Msg[#WngIndex + 28] := "A0302_PareggiatoreTesta".Warning.Centraggio.Rest_MissingExtEnable;
   "Area03_Messages".W.Msg[#WngIndex + 29] := "A0302_PareggiatoreTesta".Warning.Centraggio.Work_MissingExtEnable;
   "Area03_Messages".W.Msg[#WngIndex + 30] := "A0302_PareggiatoreTesta".Warning.Centraggio.Missing_Rest_Ls_ON[1];
   "Area03_Messages".W.Msg[#WngIndex + 31] := "A0302_PareggiatoreTesta".Warning.Centraggio.Missing_Work_Ls_ON[1];
   "Area03_Messages".W.Msg[#WngIndex + 32] := FALSE;
   "Area03_Messages".W.Msg[#WngIndex + 33] := "A0302_PareggiatoreTesta".Warning.SW_Limit_AntiCollision;
   "Area03_Messages".W.Msg[#WngIndex + 34] := "A0302_PareggiatoreTesta".Warning.MissingCnd.OP_REST_Bloccaggio;
   "Area03_Messages".W.Msg[#WngIndex + 35] := "A0302_PareggiatoreTesta".Warning.MissingCnd.OP_WORK_Bloccaggio;
   "Area03_Messages".W.Msg[#WngIndex + 36] := "A0302_PareggiatoreTesta".Warning.MissingCnd.OP_REST_Centraggio;
   "Area03_Messages".W.Msg[#WngIndex + 37] := "A0302_PareggiatoreTesta".Warning.MissingCnd.OP_WORK_Centraggio;
   "Area03_Messages".W.Msg[#WngIndex + 38] := "A0302_PareggiatoreTesta".Warning.MissingCnd.OP_REST_Sollevamento;
   "Area03_Messages".W.Msg[#WngIndex + 39] := "A0302_PareggiatoreTesta".Warning.MissingCnd.OP_WORK_Sollevamento;

   //Manipolatore
   // 
   #WngIndex := 700;

   "Area03_Messages".W.Msg[#WngIndex + 0] := "A0302_Manipolatore".Warning.Testa.Ax.NotAutReady;
   "Area03_Messages".W.Msg[#WngIndex + 1] := "A0302_Manipolatore".Warning.Testa.Ax.Minus_CndMissing;
   "Area03_Messages".W.Msg[#WngIndex + 2] := "A0302_Manipolatore".Warning.Testa.Ax.Plus_CndMissing;
   "Area03_Messages".W.Msg[#WngIndex + 3] := "A0302_Manipolatore".Warning.Testa.Ax.S120_Warning;
   "Area03_Messages".W.Msg[#WngIndex + 4] := "A0302_Manipolatore".Warning.Testa.Ax.Ax_NotHomed;
   "Area03_Messages".W.Msg[#WngIndex + 5] := "A0302_Manipolatore".Warning.Testa.Ax.Ax_FlyingHome;
   "Area03_Messages".W.Msg[#WngIndex + 6] := "A0302_Manipolatore".Warning.Testa.Ax.Ax_SwLimitMinus;
   "Area03_Messages".W.Msg[#WngIndex + 7] := "A0302_Manipolatore".Warning.Testa.Ax.Ax_SwLimitPlus;
   "Area03_Messages".W.Msg[#WngIndex + 8] := FALSE;
   "Area03_Messages".W.Msg[#WngIndex + 9] := FALSE;
   "Area03_Messages".W.Msg[#WngIndex + 10] := "A0302_Manipolatore".Warning.Testa.Sollevatore.NotAutReady;
   "Area03_Messages".W.Msg[#WngIndex + 11] := "A0302_Manipolatore".Warning.Testa.Sollevatore.PressureRunning_Timeout;
   "Area03_Messages".W.Msg[#WngIndex + 12] := "A0302_Manipolatore".Warning.Testa.Sollevatore.Rest_MissingExtEnable;
   "Area03_Messages".W.Msg[#WngIndex + 13] := "A0302_Manipolatore".Warning.Testa.Sollevatore.Work_MissingExtEnable;
   "Area03_Messages".W.Msg[#WngIndex + 14] := "A0302_Manipolatore".Warning.Testa.Sollevatore.Missing_Rest_Ls_ON[1];
   "Area03_Messages".W.Msg[#WngIndex + 15] := "A0302_Manipolatore".Warning.Testa.Sollevatore.Missing_Work_Ls_ON[1];
   "Area03_Messages".W.Msg[#WngIndex + 16] := FALSE;
   "Area03_Messages".W.Msg[#WngIndex + 17] := FALSE;
   "Area03_Messages".W.Msg[#WngIndex + 18] := "A0302_Manipolatore".Warning.Testa.Magnete.NotAutReady;
   "Area03_Messages".W.Msg[#WngIndex + 19] := "A0302_Manipolatore".Warning.Testa.Magnete.PressureRunning_Timeout;
   "Area03_Messages".W.Msg[#WngIndex + 20] := "A0302_Manipolatore".Warning.Testa.Magnete.Rest_MissingExtEnable;
   "Area03_Messages".W.Msg[#WngIndex + 21] := "A0302_Manipolatore".Warning.Testa.Magnete.Work_MissingExtEnable;
   "Area03_Messages".W.Msg[#WngIndex + 22] := "A0302_Manipolatore".Warning.Testa.Magnete.Missing_Rest_Ls_ON[1];
   "Area03_Messages".W.Msg[#WngIndex + 23] := "A0302_Manipolatore".Warning.Testa.Magnete.Missing_Work_Ls_ON[1];
   "Area03_Messages".W.Msg[#WngIndex + 24] := FALSE;
   "Area03_Messages".W.Msg[#WngIndex + 25] := FALSE;
   "Area03_Messages".W.Msg[#WngIndex + 26] := "A0302_Manipolatore".Warning.Coda.Ax.NotAutReady;
   "Area03_Messages".W.Msg[#WngIndex + 27] := "A0302_Manipolatore".Warning.Coda.Ax.Minus_CndMissing;
   "Area03_Messages".W.Msg[#WngIndex + 28] := "A0302_Manipolatore".Warning.Coda.Ax.Plus_CndMissing;
   "Area03_Messages".W.Msg[#WngIndex + 29] := "A0302_Manipolatore".Warning.Coda.Ax.S120_Warning;
   "Area03_Messages".W.Msg[#WngIndex + 30] := "A0302_Manipolatore".Warning.Coda.Ax.Ax_NotHomed;
   "Area03_Messages".W.Msg[#WngIndex + 31] := "A0302_Manipolatore".Warning.Coda.Ax.Ax_FlyingHome;
   "Area03_Messages".W.Msg[#WngIndex + 32] := "A0302_Manipolatore".Warning.Coda.Ax.Ax_SwLimitMinus;
   "Area03_Messages".W.Msg[#WngIndex + 33] := "A0302_Manipolatore".Warning.Coda.Ax.Ax_SwLimitPlus;
   "Area03_Messages".W.Msg[#WngIndex + 34] := FALSE;
   "Area03_Messages".W.Msg[#WngIndex + 35] := FALSE;
   "Area03_Messages".W.Msg[#WngIndex + 36] := "A0302_Manipolatore".Warning.Coda.Sollevatore.NotAutReady;
   "Area03_Messages".W.Msg[#WngIndex + 37] := "A0302_Manipolatore".Warning.Coda.Sollevatore.PressureRunning_Timeout;
   "Area03_Messages".W.Msg[#WngIndex + 38] := "A0302_Manipolatore".Warning.Coda.Sollevatore.Rest_MissingExtEnable;
   "Area03_Messages".W.Msg[#WngIndex + 39] := "A0302_Manipolatore".Warning.Coda.Sollevatore.Work_MissingExtEnable;
   "Area03_Messages".W.Msg[#WngIndex + 40] := "A0302_Manipolatore".Warning.Coda.Sollevatore.Missing_Rest_Ls_ON[1];
   "Area03_Messages".W.Msg[#WngIndex + 41] := "A0302_Manipolatore".Warning.Coda.Sollevatore.Missing_Work_Ls_ON[1];
   "Area03_Messages".W.Msg[#WngIndex + 42] := FALSE;
   "Area03_Messages".W.Msg[#WngIndex + 43] := FALSE;
   "Area03_Messages".W.Msg[#WngIndex + 44] := "A0302_Manipolatore".Warning.Testa.Magnete.NotAutReady;
   "Area03_Messages".W.Msg[#WngIndex + 45] := "A0302_Manipolatore".Warning.Testa.Magnete.PressureRunning_Timeout;
   "Area03_Messages".W.Msg[#WngIndex + 46] := "A0302_Manipolatore".Warning.Testa.Magnete.Rest_MissingExtEnable;
   "Area03_Messages".W.Msg[#WngIndex + 47] := "A0302_Manipolatore".Warning.Testa.Magnete.Work_MissingExtEnable;
   "Area03_Messages".W.Msg[#WngIndex + 48] := "A0302_Manipolatore".Warning.Testa.Magnete.Missing_Rest_Ls_ON[1];
   "Area03_Messages".W.Msg[#WngIndex + 49] := "A0302_Manipolatore".Warning.Testa.Magnete.Missing_Work_Ls_ON[1];
   "Area03_Messages".W.Msg[#WngIndex + 50] := "A0302_Manipolatore".Warning.MissingCnd.OP_REST_Sollevamento;
   "Area03_Messages".W.Msg[#WngIndex + 51] := "A0302_Manipolatore".Warning.MissingCnd.OP_WORK_Sollevamento;
   "Area03_Messages".W.Msg[#WngIndex + 52] := "A0302_Manipolatore".Warning.MissingCnd.OP_REST_Magneti;
   "Area03_Messages".W.Msg[#WngIndex + 53] := "A0302_Manipolatore".Warning.MissingCnd.OP_WORK_Magneti;

   //Regolazione Bordatrice
   // 
   #WngIndex := 760;

   "Area03_Messages".W.Msg[#WngIndex + 0] := "A0302_Bordatrice_RegolazioneFormato".Warning.Ax_D[1].NotAutReady;
   "Area03_Messages".W.Msg[#WngIndex + 1] := "A0302_Bordatrice_RegolazioneFormato".Warning.Ax_D[1].MissingCnd_Minus;
   "Area03_Messages".W.Msg[#WngIndex + 2] := "A0302_Bordatrice_RegolazioneFormato".Warning.Ax_D[1].MissingCnd_Plus;
   "Area03_Messages".W.Msg[#WngIndex + 3] := "A0302_Bordatrice_RegolazioneFormato".Warning.Ax_D[1].Ax_NotHomed;
   "Area03_Messages".W.Msg[#WngIndex + 4] := "A0302_Bordatrice_RegolazioneFormato".Warning.Ax_D[1].Ax.SwLimitMinus;
   "Area03_Messages".W.Msg[#WngIndex + 5] := "A0302_Bordatrice_RegolazioneFormato".Warning.Ax_D[1].Ax.SwLimitPlus;
   "Area03_Messages".W.Msg[#WngIndex + 6] := "A0302_Bordatrice_RegolazioneFormato".Warning.Ax_D[1].S120.Drive;
   "Area03_Messages".W.Msg[#WngIndex + 7] := FALSE;
   "Area03_Messages".W.Msg[#WngIndex + 8] := "A0302_Bordatrice_RegolazioneFormato".Warning.Ax_M[1].NotAutReady;
   "Area03_Messages".W.Msg[#WngIndex + 9] := "A0302_Bordatrice_RegolazioneFormato".Warning.Ax_M[1].Minus_CndMissing;
   "Area03_Messages".W.Msg[#WngIndex + 10] := "A0302_Bordatrice_RegolazioneFormato".Warning.Ax_M[1].Plus_CndMissing;
   "Area03_Messages".W.Msg[#WngIndex + 11] := "A0302_Bordatrice_RegolazioneFormato".Warning.Ax_M[1].Ax_NotHomed;
   "Area03_Messages".W.Msg[#WngIndex + 12] := "A0302_Bordatrice_RegolazioneFormato".Warning.Ax_M[1].Ax.SwLimitMinus;
   "Area03_Messages".W.Msg[#WngIndex + 13] := "A0302_Bordatrice_RegolazioneFormato".Warning.Ax_M[1].Ax.SwLimitPlus;
   "Area03_Messages".W.Msg[#WngIndex + 14] := "A0302_Bordatrice_RegolazioneFormato".Warning.Ax_M[2].NotAutReady;
   "Area03_Messages".W.Msg[#WngIndex + 15] := "A0302_Bordatrice_RegolazioneFormato".Warning.Ax_M[2].Minus_CndMissing;
   "Area03_Messages".W.Msg[#WngIndex + 16] := "A0302_Bordatrice_RegolazioneFormato".Warning.Ax_M[2].Plus_CndMissing;
   "Area03_Messages".W.Msg[#WngIndex + 17] := "A0302_Bordatrice_RegolazioneFormato".Warning.Ax_M[2].Ax_NotHomed;
   "Area03_Messages".W.Msg[#WngIndex + 18] := "A0302_Bordatrice_RegolazioneFormato".Warning.Ax_M[2].Ax.SwLimitMinus;
   "Area03_Messages".W.Msg[#WngIndex + 19] := "A0302_Bordatrice_RegolazioneFormato".Warning.Ax_M[2].Ax.SwLimitPlus;
   "Area03_Messages".W.Msg[#WngIndex + 20] := "A0302_Bordatrice_RegolazioneFormato".Warning.Ax_M[3].NotAutReady;
   "Area03_Messages".W.Msg[#WngIndex + 21] := "A0302_Bordatrice_RegolazioneFormato".Warning.Ax_M[3].Minus_CndMissing;
   "Area03_Messages".W.Msg[#WngIndex + 22] := "A0302_Bordatrice_RegolazioneFormato".Warning.Ax_M[3].Plus_CndMissing;
   "Area03_Messages".W.Msg[#WngIndex + 23] := "A0302_Bordatrice_RegolazioneFormato".Warning.Ax_M[3].Ax_NotHomed;
   "Area03_Messages".W.Msg[#WngIndex + 24] := "A0302_Bordatrice_RegolazioneFormato".Warning.Ax_M[3].Ax.SwLimitMinus;
   "Area03_Messages".W.Msg[#WngIndex + 25] := "A0302_Bordatrice_RegolazioneFormato".Warning.Ax_M[3].Ax.SwLimitPlus;
   "Area03_Messages".W.Msg[#WngIndex + 26] := "A0302_Bordatrice_RegolazioneFormato".Warning.Ax_M[4].NotAutReady;
   "Area03_Messages".W.Msg[#WngIndex + 27] := "A0302_Bordatrice_RegolazioneFormato".Warning.Ax_M[4].Minus_CndMissing;
   "Area03_Messages".W.Msg[#WngIndex + 28] := "A0302_Bordatrice_RegolazioneFormato".Warning.Ax_M[4].Plus_CndMissing;
   "Area03_Messages".W.Msg[#WngIndex + 29] := "A0302_Bordatrice_RegolazioneFormato".Warning.Ax_M[4].Ax_NotHomed;
   "Area03_Messages".W.Msg[#WngIndex + 30] := "A0302_Bordatrice_RegolazioneFormato".Warning.Ax_M[4].Ax.SwLimitMinus;
   "Area03_Messages".W.Msg[#WngIndex + 31] := "A0302_Bordatrice_RegolazioneFormato".Warning.Ax_M[4].Ax.SwLimitPlus;
   "Area03_Messages".W.Msg[#WngIndex + 32] := "A0302_Bordatrice_RegolazioneFormato".Warning.Ax_M[5].NotAutReady;
   "Area03_Messages".W.Msg[#WngIndex + 33] := "A0302_Bordatrice_RegolazioneFormato".Warning.Ax_M[5].Minus_CndMissing;
   "Area03_Messages".W.Msg[#WngIndex + 34] := "A0302_Bordatrice_RegolazioneFormato".Warning.Ax_M[5].Plus_CndMissing;
   "Area03_Messages".W.Msg[#WngIndex + 35] := "A0302_Bordatrice_RegolazioneFormato".Warning.Ax_M[5].Ax_NotHomed;
   "Area03_Messages".W.Msg[#WngIndex + 36] := "A0302_Bordatrice_RegolazioneFormato".Warning.Ax_M[5].Ax.SwLimitMinus;
   "Area03_Messages".W.Msg[#WngIndex + 37] := "A0302_Bordatrice_RegolazioneFormato".Warning.Ax_M[5].Ax.SwLimitPlus;
   "Area03_Messages".W.Msg[#WngIndex + 38] := "A0302_Bordatrice_RegolazioneFormato".Warning.Ax_M[6].NotAutReady;
   "Area03_Messages".W.Msg[#WngIndex + 39] := "A0302_Bordatrice_RegolazioneFormato".Warning.Ax_M[6].Minus_CndMissing;
   "Area03_Messages".W.Msg[#WngIndex + 40] := "A0302_Bordatrice_RegolazioneFormato".Warning.Ax_M[6].Plus_CndMissing;
   "Area03_Messages".W.Msg[#WngIndex + 41] := "A0302_Bordatrice_RegolazioneFormato".Warning.Ax_M[6].Ax_NotHomed;
   "Area03_Messages".W.Msg[#WngIndex + 42] := "A0302_Bordatrice_RegolazioneFormato".Warning.Ax_M[6].Ax.SwLimitMinus;
   "Area03_Messages".W.Msg[#WngIndex + 43] := "A0302_Bordatrice_RegolazioneFormato".Warning.Ax_M[6].Ax.SwLimitPlus;
   "Area03_Messages".W.Msg[#WngIndex + 44] := "A0302_Bordatrice_RegolazioneFormato".Warning.Ax_M[7].NotAutReady;
   "Area03_Messages".W.Msg[#WngIndex + 45] := "A0302_Bordatrice_RegolazioneFormato".Warning.Ax_M[7].Minus_CndMissing;
   "Area03_Messages".W.Msg[#WngIndex + 46] := "A0302_Bordatrice_RegolazioneFormato".Warning.Ax_M[7].Plus_CndMissing;
   "Area03_Messages".W.Msg[#WngIndex + 47] := "A0302_Bordatrice_RegolazioneFormato".Warning.Ax_M[7].Ax_NotHomed;
   "Area03_Messages".W.Msg[#WngIndex + 48] := "A0302_Bordatrice_RegolazioneFormato".Warning.Ax_M[7].Ax.SwLimitMinus;
   "Area03_Messages".W.Msg[#WngIndex + 49] := "A0302_Bordatrice_RegolazioneFormato".Warning.Ax_M[7].Ax.SwLimitPlus;
   "Area03_Messages".W.Msg[#WngIndex + 50] := "A0302_Bordatrice_RegolazioneFormato".Warning.Ax_M[8].NotAutReady;
   "Area03_Messages".W.Msg[#WngIndex + 51] := "A0302_Bordatrice_RegolazioneFormato".Warning.Ax_M[8].Minus_CndMissing;
   "Area03_Messages".W.Msg[#WngIndex + 52] := "A0302_Bordatrice_RegolazioneFormato".Warning.Ax_M[8].Plus_CndMissing;
   "Area03_Messages".W.Msg[#WngIndex + 53] := "A0302_Bordatrice_RegolazioneFormato".Warning.Ax_M[8].Ax_NotHomed;
   "Area03_Messages".W.Msg[#WngIndex + 54] := "A0302_Bordatrice_RegolazioneFormato".Warning.Ax_M[8].Ax.SwLimitMinus;
   "Area03_Messages".W.Msg[#WngIndex + 55] := "A0302_Bordatrice_RegolazioneFormato".Warning.Ax_M[8].Ax.SwLimitPlus;
   "Area03_Messages".W.Msg[#WngIndex + 56] := "A0302_Bordatrice_RegolazioneFormato".Warning.Ax_M[9].NotAutReady;
   "Area03_Messages".W.Msg[#WngIndex + 57] := "A0302_Bordatrice_RegolazioneFormato".Warning.Ax_M[9].Minus_CndMissing;
   "Area03_Messages".W.Msg[#WngIndex + 58] := "A0302_Bordatrice_RegolazioneFormato".Warning.Ax_M[9].Plus_CndMissing;
   "Area03_Messages".W.Msg[#WngIndex + 59] := "A0302_Bordatrice_RegolazioneFormato".Warning.Ax_M[9].Ax_NotHomed;
   "Area03_Messages".W.Msg[#WngIndex + 60] := "A0302_Bordatrice_RegolazioneFormato".Warning.Ax_M[9].Ax.SwLimitMinus;
   "Area03_Messages".W.Msg[#WngIndex + 61] := "A0302_Bordatrice_RegolazioneFormato".Warning.Ax_M[9].Ax.SwLimitPlus;
   "Area03_Messages".W.Msg[#WngIndex + 62] := FALSE;
   "Area03_Messages".W.Msg[#WngIndex + 63] := "A0302_Bordatrice_RegolazioneFormato".Warning.Passaggio01_MaxDisallineamentoAXs;
   "Area03_Messages".W.Msg[#WngIndex + 64] := "A0302_Bordatrice_RegolazioneFormato".Warning.Passaggio02_MaxDisallineamentoAXs;
   "Area03_Messages".W.Msg[#WngIndex + 65] := "A0302_Bordatrice_RegolazioneFormato".Warning.Passaggio03_MaxDisallineamentoAXs;
   "Area03_Messages".W.Msg[#WngIndex + 66] := "A0302_Bordatrice_RegolazioneFormato".Warning.Passaggio04_MaxDisallineamentoAXs;
   "Area03_Messages".W.Msg[#WngIndex + 67] := FALSE;
   "Area03_Messages".W.Msg[#WngIndex + 68] := FALSE;
   "Area03_Messages".W.Msg[#WngIndex + 69] := FALSE;


   // Finale 829


   (*
   "Area03_Messages".W.Msg[#WngIndex + 0] := FALSE;
   "Area03_Messages".W.Msg[#WngIndex + 1] := FALSE;
   "Area03_Messages".W.Msg[#WngIndex + 2] := FALSE;
   "Area03_Messages".W.Msg[#WngIndex + 3] := FALSE;
   "Area03_Messages".W.Msg[#WngIndex + 4] := FALSE;
   "Area03_Messages".W.Msg[#WngIndex + 5] := FALSE;
   "Area03_Messages".W.Msg[#WngIndex + 6] := FALSE;
   "Area03_Messages".W.Msg[#WngIndex + 7] := FALSE;
   "Area03_Messages".W.Msg[#WngIndex + 8] := FALSE;
   "Area03_Messages".W.Msg[#WngIndex + 9] := FALSE;
   "Area03_Messages".W.Msg[#WngIndex + 10] := FALSE;
   "Area03_Messages".W.Msg[#WngIndex + 11] := FALSE;
   "Area03_Messages".W.Msg[#WngIndex + 12] := FALSE;
   "Area03_Messages".W.Msg[#WngIndex + 13] := FALSE;
   "Area03_Messages".W.Msg[#WngIndex + 14] := FALSE;
   "Area03_Messages".W.Msg[#WngIndex + 15] := FALSE;
   "Area03_Messages".W.Msg[#WngIndex + 16] := FALSE;
   "Area03_Messages".W.Msg[#WngIndex + 17] := FALSE;
   "Area03_Messages".W.Msg[#WngIndex + 18] := FALSE;
   "Area03_Messages".W.Msg[#WngIndex + 19] := FALSE;
   "Area03_Messages".W.Msg[#WngIndex + 20] := FALSE;
   "Area03_Messages".W.Msg[#WngIndex + 21] := FALSE;
   "Area03_Messages".W.Msg[#WngIndex + 22] := FALSE;
   "Area03_Messages".W.Msg[#WngIndex + 23] := FALSE;
   "Area03_Messages".W.Msg[#WngIndex + 24] := FALSE;
   "Area03_Messages".W.Msg[#WngIndex + 25] := FALSE;
   "Area03_Messages".W.Msg[#WngIndex + 26] := FALSE;
   "Area03_Messages".W.Msg[#WngIndex + 27] := FALSE;
   "Area03_Messages".W.Msg[#WngIndex + 28] := FALSE;
   "Area03_Messages".W.Msg[#WngIndex + 29] := FALSE;
   "Area03_Messages".W.Msg[#WngIndex + 30] := FALSE;
   "Area03_Messages".W.Msg[#WngIndex + 31] := FALSE;
   "Area03_Messages".W.Msg[#WngIndex + 32] := FALSE;
   "Area03_Messages".W.Msg[#WngIndex + 33] := FALSE;
   "Area03_Messages".W.Msg[#WngIndex + 34] := FALSE;
   "Area03_Messages".W.Msg[#WngIndex + 35] := FALSE;
   "Area03_Messages".W.Msg[#WngIndex + 36] := FALSE;
   "Area03_Messages".W.Msg[#WngIndex + 37] := FALSE;
   "Area03_Messages".W.Msg[#WngIndex + 38] := FALSE;
   "Area03_Messages".W.Msg[#WngIndex + 39] := FALSE;
   *)
END_REGION

REGION Network 17: Warnings manager
   RUNG wire#powerrail
      "Area03_Msg_Warnings"(Ack := wire#w1, Messages := "Area03_Messages".W.Msg, MessagesHMI := "Area03_Messages".W.Hmi, MessagesACK := "Area03_Messages".W.Ack, MessagePresence =>, NewMessage =>, MessageCount => "A03_HMI".Area03.Status.WarningsNumber)
   END_RUNG
   RUNG wire#powerrail
      Contact( "Area03".DataIn.PbAckRst )
   END_RUNG wire#w1
   // the same network as SCL:
   "Area03_Msg_Warnings"(Ack := "Area03".DataIn.PbAckRst,   // "MsgManager"
                         Messages := "Area03_Messages".W.Msg,
                         MessagesHMI := "Area03_Messages".W.Hmi,
                         MessagesACK := "Area03_Messages".W.Ack,
                         MessageCount => "A03_HMI".Area03.Status.WarningsNumber);
END_REGION

REGION Network 19: >
END_REGION

REGION Network 20: >
END_REGION

REGION Network 21: >
END_REGION

REGION Network 22: MB lamp indicators
   RUNG wire#powerrail
      Contact( "Area03".DataOut.lampReady )
      Coil( "MB3_Lp_Abilitazione_Automatico_Area03" )
   END_RUNG
   RUNG wire#powerrail
      Contact( "Area03".DataOut.lampCycle )
      Coil( "MB3_Lp_Start_Ciclo_Area03" )
   END_RUNG
   RUNG wire#powerrail
      I_Contact( "Area03".DataOut.LampAlarmPresence )
      I_Contact( "Area03".DataOut.LampWarningPresence )
      Not()
      wire#w1
      Contact( "Sys".Clock_1S )
      wire#w2
      Coil( "MB3_Lp_Reset_Anomalie" )
   END_RUNG
   RUNG wire#w1
      I_Contact( "Area03_Msg_Alarms".NewMessage )
   END_RUNG wire#w2
   RUNG wire#powerrail
      Contact( "MB3_Pb_Avanti_Stazione_1_Area03" )
      Coil( "MB3_Lp_Avanti_Stazione_1_Area03" )
   END_RUNG
   RUNG wire#powerrail
      Contact( "MB3_Pb_Avanti_Stazione_2_Area03" )
      Coil( "MB3_Lp_Avanti_Stazione_2_Area03" )
   END_RUNG
   // the same network as SCL:
   "MB3_Lp_Abilitazione_Automatico_Area03" := "Area03".DataOut.lampReady;
   "MB3_Lp_Start_Ciclo_Area03" := "Area03".DataOut.lampCycle;
   "MB3_Lp_Reset_Anomalie" := NOT (NOT "Area03".DataOut.LampAlarmPresence AND NOT "Area03".DataOut.LampWarningPresence) AND ("Sys".Clock_1S OR NOT "Area03_Msg_Alarms".NewMessage);
   "MB3_Lp_Avanti_Stazione_1_Area03" := "MB3_Pb_Avanti_Stazione_1_Area03";
   "MB3_Lp_Avanti_Stazione_2_Area03" := "MB3_Pb_Avanti_Stazione_2_Area03";
END_REGION

REGION Network 23: Tower lamp
END_REGION

REGION Network 24: Super User
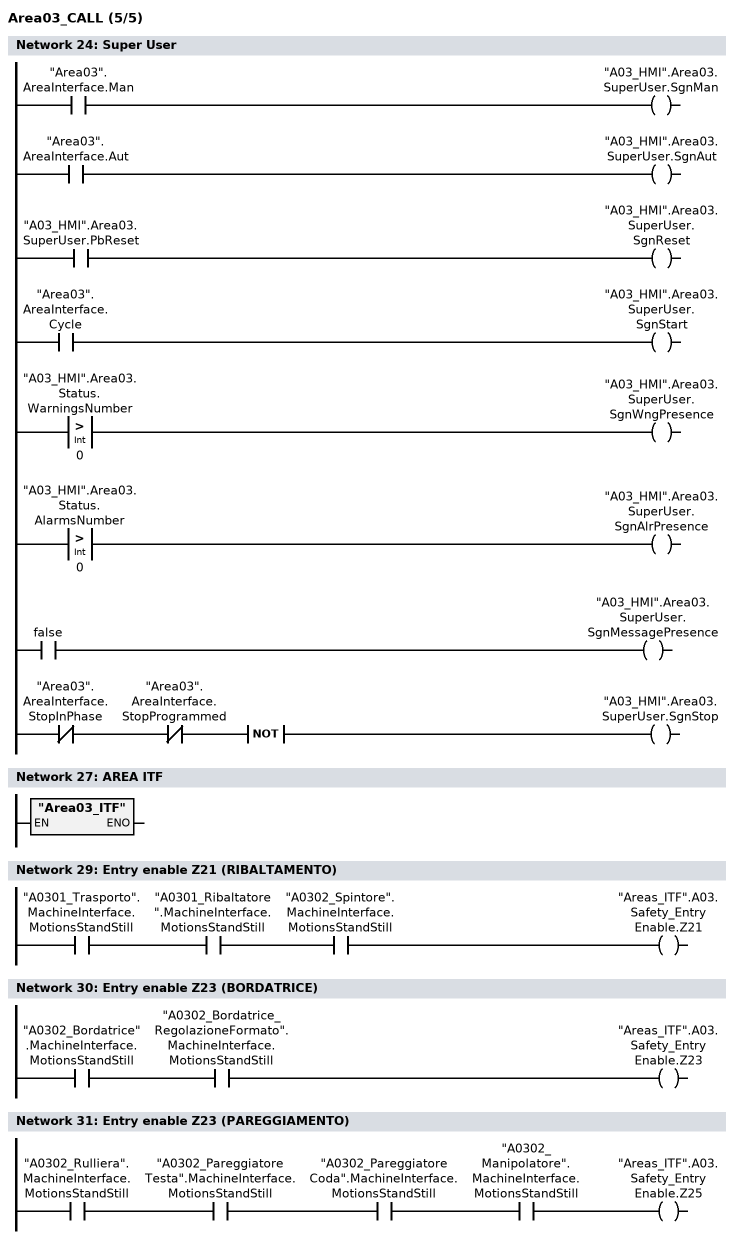
   RUNG wire#powerrail
      Contact( "Area03".AreaInterface.Man )
      Coil( "A03_HMI".Area03.SuperUser.SgnMan )
   END_RUNG
   RUNG wire#powerrail
      Contact( "Area03".AreaInterface.Aut )
      Coil( "A03_HMI".Area03.SuperUser.SgnAut )
   END_RUNG
   RUNG wire#powerrail
      Contact( "A03_HMI".Area03.SuperUser.PbReset )
      Coil( "A03_HMI".Area03.SuperUser.SgnReset )
   END_RUNG
   RUNG wire#powerrail
      Contact( "Area03".AreaInterface.Cycle )
      Coil( "A03_HMI".Area03.SuperUser.SgnStart )
   END_RUNG
   RUNG wire#powerrail
      { S7_Templates := "SrcType := Int" } GT_Contact(in1 := "A03_HMI".Area03.Status.WarningsNumber, in2 := 0)
      Coil( "A03_HMI".Area03.SuperUser.SgnWngPresence )
   END_RUNG
   RUNG wire#powerrail
      { S7_Templates := "SrcType := Int" } GT_Contact(in1 := "A03_HMI".Area03.Status.AlarmsNumber, in2 := 0)
      Coil( "A03_HMI".Area03.SuperUser.SgnAlrPresence )
   END_RUNG
   RUNG wire#powerrail
      Contact( false )
      Coil( "A03_HMI".Area03.SuperUser.SgnMessagePresence )
   END_RUNG
   RUNG wire#powerrail
      I_Contact( "Area03".AreaInterface.StopInPhase )
      I_Contact( "Area03".AreaInterface.StopProgrammed )
      Not()
      Coil( "A03_HMI".Area03.SuperUser.SgnStop )
   END_RUNG
   // the same network as SCL:
   "A03_HMI".Area03.SuperUser.SgnMan := "Area03".AreaInterface.Man;
   "A03_HMI".Area03.SuperUser.SgnAut := "Area03".AreaInterface.Aut;
   "A03_HMI".Area03.SuperUser.SgnReset := "A03_HMI".Area03.SuperUser.PbReset;
   "A03_HMI".Area03.SuperUser.SgnStart := "Area03".AreaInterface.Cycle;
   "A03_HMI".Area03.SuperUser.SgnWngPresence := "A03_HMI".Area03.Status.WarningsNumber > 0;
   "A03_HMI".Area03.SuperUser.SgnAlrPresence := "A03_HMI".Area03.Status.AlarmsNumber > 0;
   "A03_HMI".Area03.SuperUser.SgnMessagePresence := false;
   "A03_HMI".Area03.SuperUser.SgnStop := NOT (NOT "Area03".AreaInterface.StopInPhase AND NOT "Area03".AreaInterface.StopProgrammed);
END_REGION

REGION Network 25 (SCL): <<< MACHINES AREA 03 >>>
   // Gen
   "A03_HMI_CALL"();



   // A0301
   // //
   "A0301_Manager_CALL"();

   "A0301_Trasporto_CALL"();

   "A0301_Fermi_P1_CALL"();

   "A0301_Fermi_P2_CALL"();

   "A0301_Fermi_P3_CALL"();

   "A0301_Ribaltatore_CALL"();

   "A0301_Fermi_P4_CALL"();

   "A0301_Spintore_Lat_CALL"();

   //A0302
   //
   "A0302_Manager_CALL"();

   "A0302_HU_Cytropack_CALL"();

   "A0302_Spintore_CALL"();

   "A0302_Bordatrice_CALL"();

   "A0302_Bordatrice_RegolazioneFormato_OB1_CALL"();

   "A0302_Rulliera_CALL"();

   "A0302_Centratori_CALL"();

   "A0302_PareggiatoreCoda_CALL"();

   "A0302_PareggiatoreTesta_CALL"();

   "A0302_Manipolatore_CALL"();



   "A03_TrkManager_CALL"();
END_REGION

REGION Network 26: >
END_REGION

REGION Network 27: AREA ITF
   RUNG wire#powerrail
      "Area03_ITF"()
   END_RUNG
   // the same network as SCL:
   "Area03_ITF"();
END_REGION

REGION Network 28: >
END_REGION

REGION Network 29: Entry enable Z21 (RIBALTAMENTO)
   RUNG wire#powerrail
      Contact( "A0301_Trasporto".MachineInterface.MotionsStandStill )
      Contact( "A0301_Ribaltatore".MachineInterface.MotionsStandStill )
      Contact( "A0302_Spintore".MachineInterface.MotionsStandStill )
      Coil( "Areas_ITF".A03.Safety_EntryEnable.Z21 )
   END_RUNG
   // the same network as SCL:
   "Areas_ITF".A03.Safety_EntryEnable.Z21 := "A0301_Trasporto".MachineInterface.MotionsStandStill AND "A0301_Ribaltatore".MachineInterface.MotionsStandStill AND "A0302_Spintore".MachineInterface.MotionsStandStill;
END_REGION

REGION Network 30: Entry enable Z23 (BORDATRICE)
   RUNG wire#powerrail
      Contact( "A0302_Bordatrice".MachineInterface.MotionsStandStill )
      Contact( "A0302_Bordatrice_RegolazioneFormato".MachineInterface.MotionsStandStill )
      Coil( "Areas_ITF".A03.Safety_EntryEnable.Z23 )
   END_RUNG
   // the same network as SCL:
   "Areas_ITF".A03.Safety_EntryEnable.Z23 := "A0302_Bordatrice".MachineInterface.MotionsStandStill AND "A0302_Bordatrice_RegolazioneFormato".MachineInterface.MotionsStandStill;
END_REGION

REGION Network 31: Entry enable Z23 (PAREGGIAMENTO)
   RUNG wire#powerrail
      Contact( "A0302_Rulliera".MachineInterface.MotionsStandStill )
      Contact( "A0302_PareggiatoreTesta".MachineInterface.MotionsStandStill )
      Contact( "A0302_PareggiatoreCoda".MachineInterface.MotionsStandStill )
      Contact( "A0302_Manipolatore".MachineInterface.MotionsStandStill )
      Coil( "Areas_ITF".A03.Safety_EntryEnable.Z25 )
   END_RUNG
   // the same network as SCL:
   "Areas_ITF".A03.Safety_EntryEnable.Z25 := "A0302_Rulliera".MachineInterface.MotionsStandStill AND "A0302_PareggiatoreTesta".MachineInterface.MotionsStandStill AND "A0302_PareggiatoreCoda".MachineInterface.MotionsStandStill AND "A0302_Manipolatore".MachineInterface.MotionsStandStill;
END_REGION

REGION Network 32: >
END_REGION
END_FUNCTION

FUNCTION "Area03_ITF" : Void   // FC22, LAD
// stored: SetENOAutomatically false
BEGIN

REGION Network 2: AREA ITF
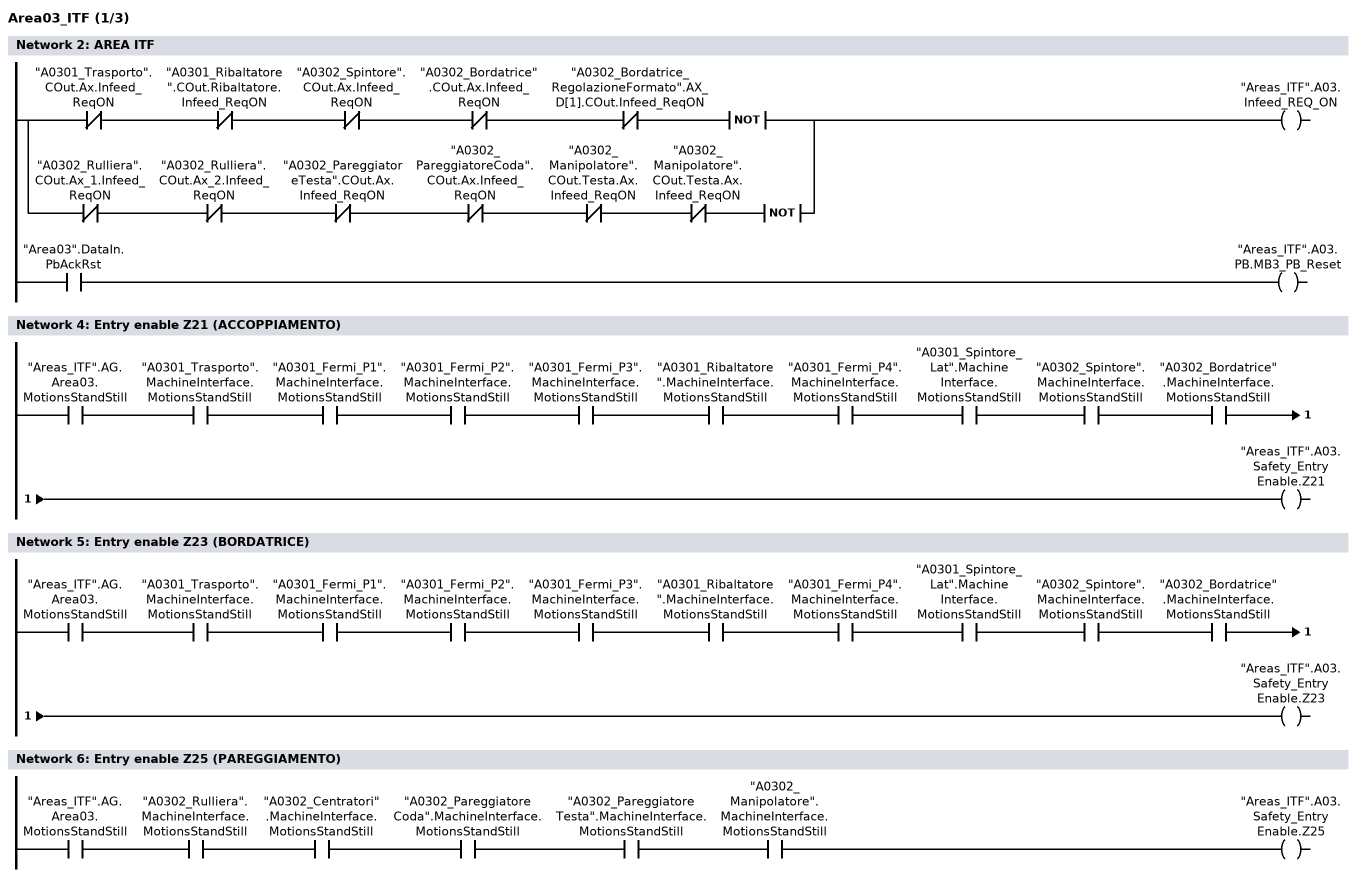
   RUNG wire#powerrail
      I_Contact( "A0301_Trasporto".COut.Ax.Infeed_ReqON )
      I_Contact( "A0301_Ribaltatore".COut.Ribaltatore.Infeed_ReqON )
      I_Contact( "A0302_Spintore".COut.Ax.Infeed_ReqON )
      I_Contact( "A0302_Bordatrice".COut.Ax.Infeed_ReqON )
      I_Contact( "A0302_Bordatrice_RegolazioneFormato".AX_D[1].COut.Infeed_ReqON )
      Not()
      wire#w1
      Coil( "Areas_ITF".A03.Infeed_REQ_ON )
   END_RUNG
   RUNG wire#powerrail
      I_Contact( "A0302_Rulliera".COut.Ax_1.Infeed_ReqON )
      I_Contact( "A0302_Rulliera".COut.Ax_2.Infeed_ReqON )
      I_Contact( "A0302_PareggiatoreTesta".COut.Ax.Infeed_ReqON )
      I_Contact( "A0302_PareggiatoreCoda".COut.Ax.Infeed_ReqON )
      I_Contact( "A0302_Manipolatore".COut.Testa.Ax.Infeed_ReqON )
      I_Contact( "A0302_Manipolatore".COut.Testa.Ax.Infeed_ReqON )
      Not()
   END_RUNG wire#w1
   RUNG wire#powerrail
      Contact( "Area03".DataIn.PbAckRst )
      Coil( "Areas_ITF".A03.PB.MB3_PB_Reset )
   END_RUNG
   // the same network as SCL:
   "Areas_ITF".A03.Infeed_REQ_ON := NOT (NOT "A0301_Trasporto".COut.Ax.Infeed_ReqON AND NOT "A0301_Ribaltatore".COut.Ribaltatore.Infeed_ReqON AND NOT "A0302_Spintore".COut.Ax.Infeed_ReqON AND NOT "A0302_Bordatrice".COut.Ax.Infeed_ReqON AND NOT "A0302_Bordatrice_RegolazioneFormato".AX_D[1].COut.Infeed_ReqON) OR NOT (NOT "A0302_Rulliera".COut.Ax_1.Infeed_ReqON AND NOT "A0302_Rulliera".COut.Ax_2.Infeed_ReqON AND NOT "A0302_PareggiatoreTesta".COut.Ax.Infeed_ReqON AND NOT "A0302_PareggiatoreCoda".COut.Ax.Infeed_ReqON AND NOT "A0302_Manipolatore".COut.Testa.Ax.Infeed_ReqON AND NOT "A0302_Manipolatore".COut.Testa.Ax.Infeed_ReqON);
   "Areas_ITF".A03.PB.MB3_PB_Reset := "Area03".DataIn.PbAckRst;
END_REGION

REGION Network 3: >
END_REGION

REGION Network 4: Entry enable Z21 (ACCOPPIAMENTO)
   RUNG wire#powerrail
      Contact( "Areas_ITF".AG.Area03.MotionsStandStill )
      Contact( "A0301_Trasporto".MachineInterface.MotionsStandStill )
      Contact( "A0301_Fermi_P1".MachineInterface.MotionsStandStill )
      Contact( "A0301_Fermi_P2".MachineInterface.MotionsStandStill )
      Contact( "A0301_Fermi_P3".MachineInterface.MotionsStandStill )
      Contact( "A0301_Ribaltatore".MachineInterface.MotionsStandStill )
      Contact( "A0301_Fermi_P4".MachineInterface.MotionsStandStill )
      Contact( "A0301_Spintore_Lat".MachineInterface.MotionsStandStill )
      Contact( "A0302_Spintore".MachineInterface.MotionsStandStill )
      Contact( "A0302_Bordatrice".MachineInterface.MotionsStandStill )
      Coil( "Areas_ITF".A03.Safety_EntryEnable.Z21 )
   END_RUNG
   // the same network as SCL:
   "Areas_ITF".A03.Safety_EntryEnable.Z21 := "Areas_ITF".AG.Area03.MotionsStandStill AND "A0301_Trasporto".MachineInterface.MotionsStandStill AND "A0301_Fermi_P1".MachineInterface.MotionsStandStill AND "A0301_Fermi_P2".MachineInterface.MotionsStandStill AND "A0301_Fermi_P3".MachineInterface.MotionsStandStill AND "A0301_Ribaltatore".MachineInterface.MotionsStandStill AND "A0301_Fermi_P4".MachineInterface.MotionsStandStill AND "A0301_Spintore_Lat".MachineInterface.MotionsStandStill AND "A0302_Spintore".MachineInterface.MotionsStandStill AND "A0302_Bordatrice".MachineInterface.MotionsStandStill;
END_REGION

REGION Network 5: Entry enable Z23 (BORDATRICE)
   RUNG wire#powerrail
      Contact( "Areas_ITF".AG.Area03.MotionsStandStill )
      Contact( "A0301_Trasporto".MachineInterface.MotionsStandStill )
      Contact( "A0301_Fermi_P1".MachineInterface.MotionsStandStill )
      Contact( "A0301_Fermi_P2".MachineInterface.MotionsStandStill )
      Contact( "A0301_Fermi_P3".MachineInterface.MotionsStandStill )
      Contact( "A0301_Ribaltatore".MachineInterface.MotionsStandStill )
      Contact( "A0301_Fermi_P4".MachineInterface.MotionsStandStill )
      Contact( "A0301_Spintore_Lat".MachineInterface.MotionsStandStill )
      Contact( "A0302_Spintore".MachineInterface.MotionsStandStill )
      Contact( "A0302_Bordatrice".MachineInterface.MotionsStandStill )
      Coil( "Areas_ITF".A03.Safety_EntryEnable.Z23 )
   END_RUNG
   // the same network as SCL:
   "Areas_ITF".A03.Safety_EntryEnable.Z23 := "Areas_ITF".AG.Area03.MotionsStandStill AND "A0301_Trasporto".MachineInterface.MotionsStandStill AND "A0301_Fermi_P1".MachineInterface.MotionsStandStill AND "A0301_Fermi_P2".MachineInterface.MotionsStandStill AND "A0301_Fermi_P3".MachineInterface.MotionsStandStill AND "A0301_Ribaltatore".MachineInterface.MotionsStandStill AND "A0301_Fermi_P4".MachineInterface.MotionsStandStill AND "A0301_Spintore_Lat".MachineInterface.MotionsStandStill AND "A0302_Spintore".MachineInterface.MotionsStandStill AND "A0302_Bordatrice".MachineInterface.MotionsStandStill;
END_REGION

REGION Network 6: Entry enable Z25 (PAREGGIAMENTO)
   RUNG wire#powerrail
      Contact( "Areas_ITF".AG.Area03.MotionsStandStill )
      Contact( "A0302_Rulliera".MachineInterface.MotionsStandStill )
      Contact( "A0302_Centratori".MachineInterface.MotionsStandStill )
      Contact( "A0302_PareggiatoreCoda".MachineInterface.MotionsStandStill )
      Contact( "A0302_PareggiatoreTesta".MachineInterface.MotionsStandStill )
      Contact( "A0302_Manipolatore".MachineInterface.MotionsStandStill )
      Coil( "Areas_ITF".A03.Safety_EntryEnable.Z25 )
   END_RUNG
   // the same network as SCL:
   "Areas_ITF".A03.Safety_EntryEnable.Z25 := "Areas_ITF".AG.Area03.MotionsStandStill AND "A0302_Rulliera".MachineInterface.MotionsStandStill AND "A0302_Centratori".MachineInterface.MotionsStandStill AND "A0302_PareggiatoreCoda".MachineInterface.MotionsStandStill AND "A0302_PareggiatoreTesta".MachineInterface.MotionsStandStill AND "A0302_Manipolatore".MachineInterface.MotionsStandStill;
END_REGION

REGION Network 7: < < < < CTRL SAFE > > > >
END_REGION

REGION Network 8: Ctrl Safe S120
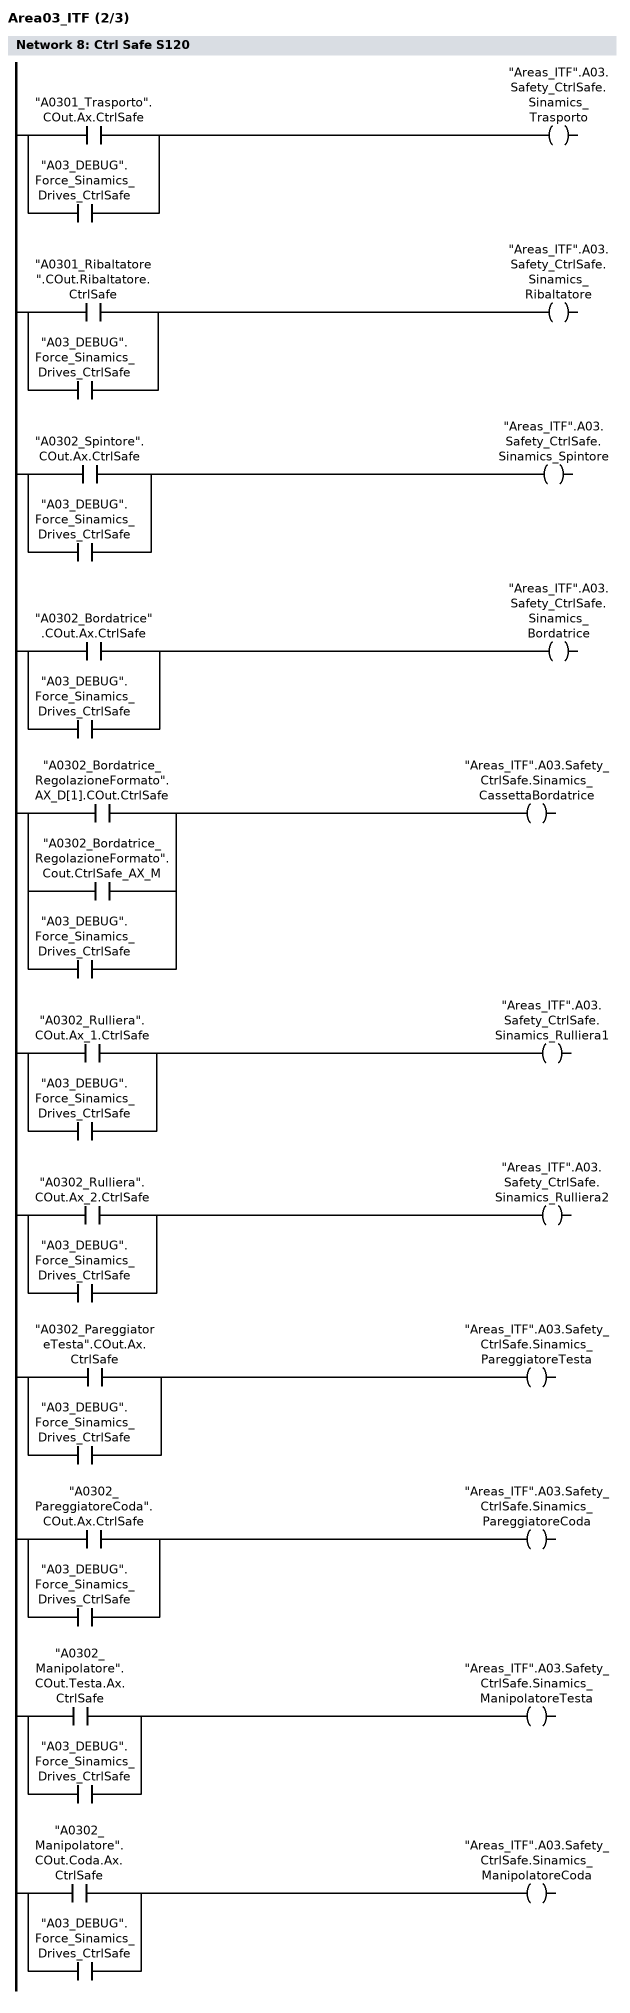
   RUNG wire#powerrail
      Contact( "A0301_Trasporto".COut.Ax.CtrlSafe )
      wire#w1
      Coil( "Areas_ITF".A03.Safety_CtrlSafe.Sinamics_Trasporto )
   END_RUNG
   RUNG wire#powerrail
      Contact( "A03_DEBUG".Force_Sinamics_Drives_CtrlSafe )
   END_RUNG wire#w1
   RUNG wire#powerrail
      Contact( "A0301_Ribaltatore".COut.Ribaltatore.CtrlSafe )
      wire#w2
      Coil( "Areas_ITF".A03.Safety_CtrlSafe.Sinamics_Ribaltatore )
   END_RUNG
   RUNG wire#powerrail
      Contact( "A03_DEBUG".Force_Sinamics_Drives_CtrlSafe )
   END_RUNG wire#w2
   RUNG wire#powerrail
      Contact( "A0302_Spintore".COut.Ax.CtrlSafe )
      wire#w3
      Coil( "Areas_ITF".A03.Safety_CtrlSafe.Sinamics_Spintore )
   END_RUNG
   RUNG wire#powerrail
      Contact( "A03_DEBUG".Force_Sinamics_Drives_CtrlSafe )
   END_RUNG wire#w3
   RUNG wire#powerrail
      Contact( "A0302_Bordatrice".COut.Ax.CtrlSafe )
      wire#w4
      Coil( "Areas_ITF".A03.Safety_CtrlSafe.Sinamics_Bordatrice )
   END_RUNG
   RUNG wire#powerrail
      Contact( "A03_DEBUG".Force_Sinamics_Drives_CtrlSafe )
   END_RUNG wire#w4
   RUNG wire#powerrail
      Contact( "A0302_Bordatrice_RegolazioneFormato".AX_D[1].COut.CtrlSafe )
      wire#w5
      Coil( "Areas_ITF".A03.Safety_CtrlSafe.Sinamics_CassettaBordatrice )
   END_RUNG
   RUNG wire#powerrail
      Contact( "A0302_Bordatrice_RegolazioneFormato".Cout.CtrlSafe_AX_M )
   END_RUNG wire#w5
   RUNG wire#powerrail
      Contact( "A03_DEBUG".Force_Sinamics_Drives_CtrlSafe )
   END_RUNG wire#w5
   RUNG wire#powerrail
      Contact( "A0302_Rulliera".COut.Ax_1.CtrlSafe )
      wire#w6
      Coil( "Areas_ITF".A03.Safety_CtrlSafe.Sinamics_Rulliera1 )
   END_RUNG
   RUNG wire#powerrail
      Contact( "A03_DEBUG".Force_Sinamics_Drives_CtrlSafe )
   END_RUNG wire#w6
   RUNG wire#powerrail
      Contact( "A0302_Rulliera".COut.Ax_2.CtrlSafe )
      wire#w7
      Coil( "Areas_ITF".A03.Safety_CtrlSafe.Sinamics_Rulliera2 )
   END_RUNG
   RUNG wire#powerrail
      Contact( "A03_DEBUG".Force_Sinamics_Drives_CtrlSafe )
   END_RUNG wire#w7
   RUNG wire#powerrail
      Contact( "A0302_PareggiatoreTesta".COut.Ax.CtrlSafe )
      wire#w8
      Coil( "Areas_ITF".A03.Safety_CtrlSafe.Sinamics_PareggiatoreTesta )
   END_RUNG
   RUNG wire#powerrail
      Contact( "A03_DEBUG".Force_Sinamics_Drives_CtrlSafe )
   END_RUNG wire#w8
   RUNG wire#powerrail
      Contact( "A0302_PareggiatoreCoda".COut.Ax.CtrlSafe )
      wire#w9
      Coil( "Areas_ITF".A03.Safety_CtrlSafe.Sinamics_PareggiatoreCoda )
   END_RUNG
   RUNG wire#powerrail
      Contact( "A03_DEBUG".Force_Sinamics_Drives_CtrlSafe )
   END_RUNG wire#w9
   RUNG wire#powerrail
      Contact( "A0302_Manipolatore".COut.Testa.Ax.CtrlSafe )
      wire#w10
      Coil( "Areas_ITF".A03.Safety_CtrlSafe.Sinamics_ManipolatoreTesta )
   END_RUNG
   RUNG wire#powerrail
      Contact( "A03_DEBUG".Force_Sinamics_Drives_CtrlSafe )
   END_RUNG wire#w10
   RUNG wire#powerrail
      Contact( "A0302_Manipolatore".COut.Coda.Ax.CtrlSafe )
      wire#w11
      Coil( "Areas_ITF".A03.Safety_CtrlSafe.Sinamics_ManipolatoreCoda )
   END_RUNG
   RUNG wire#powerrail
      Contact( "A03_DEBUG".Force_Sinamics_Drives_CtrlSafe )
   END_RUNG wire#w11
   // the same network as SCL:
   "Areas_ITF".A03.Safety_CtrlSafe.Sinamics_Trasporto := "A0301_Trasporto".COut.Ax.CtrlSafe OR "A03_DEBUG".Force_Sinamics_Drives_CtrlSafe;
   "Areas_ITF".A03.Safety_CtrlSafe.Sinamics_Ribaltatore := "A0301_Ribaltatore".COut.Ribaltatore.CtrlSafe OR "A03_DEBUG".Force_Sinamics_Drives_CtrlSafe;
   "Areas_ITF".A03.Safety_CtrlSafe.Sinamics_Spintore := "A0302_Spintore".COut.Ax.CtrlSafe OR "A03_DEBUG".Force_Sinamics_Drives_CtrlSafe;
   "Areas_ITF".A03.Safety_CtrlSafe.Sinamics_Bordatrice := "A0302_Bordatrice".COut.Ax.CtrlSafe OR "A03_DEBUG".Force_Sinamics_Drives_CtrlSafe;
   "Areas_ITF".A03.Safety_CtrlSafe.Sinamics_CassettaBordatrice := "A0302_Bordatrice_RegolazioneFormato".AX_D[1].COut.CtrlSafe OR "A0302_Bordatrice_RegolazioneFormato".Cout.CtrlSafe_AX_M OR "A03_DEBUG".Force_Sinamics_Drives_CtrlSafe;
   "Areas_ITF".A03.Safety_CtrlSafe.Sinamics_Rulliera1 := "A0302_Rulliera".COut.Ax_1.CtrlSafe OR "A03_DEBUG".Force_Sinamics_Drives_CtrlSafe;
   "Areas_ITF".A03.Safety_CtrlSafe.Sinamics_Rulliera2 := "A0302_Rulliera".COut.Ax_2.CtrlSafe OR "A03_DEBUG".Force_Sinamics_Drives_CtrlSafe;
   "Areas_ITF".A03.Safety_CtrlSafe.Sinamics_PareggiatoreTesta := "A0302_PareggiatoreTesta".COut.Ax.CtrlSafe OR "A03_DEBUG".Force_Sinamics_Drives_CtrlSafe;
   "Areas_ITF".A03.Safety_CtrlSafe.Sinamics_PareggiatoreCoda := "A0302_PareggiatoreCoda".COut.Ax.CtrlSafe OR "A03_DEBUG".Force_Sinamics_Drives_CtrlSafe;
   "Areas_ITF".A03.Safety_CtrlSafe.Sinamics_ManipolatoreTesta := "A0302_Manipolatore".COut.Testa.Ax.CtrlSafe OR "A03_DEBUG".Force_Sinamics_Drives_CtrlSafe;
   "Areas_ITF".A03.Safety_CtrlSafe.Sinamics_ManipolatoreCoda := "A0302_Manipolatore".COut.Coda.Ax.CtrlSafe OR "A03_DEBUG".Force_Sinamics_Drives_CtrlSafe;
END_REGION

REGION Network 9: Ctrl Safe Safety Valve
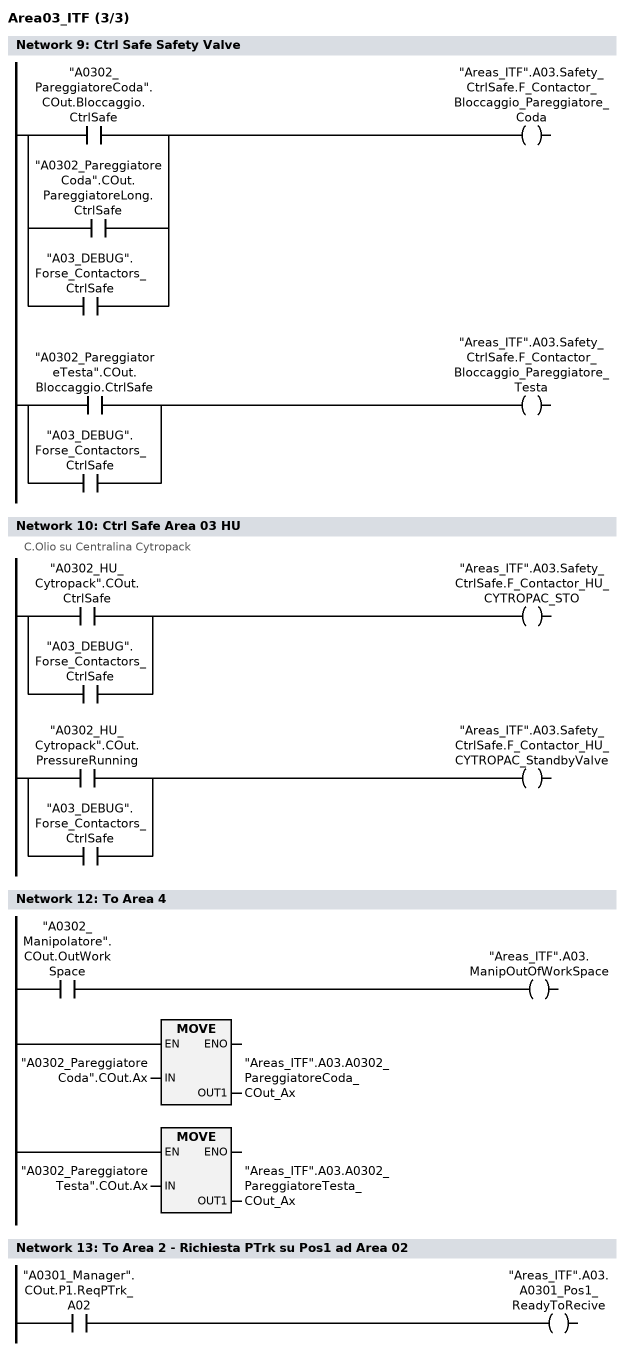
   RUNG wire#powerrail
      Contact( "A0302_PareggiatoreCoda".COut.Bloccaggio.CtrlSafe )
      wire#w1
      Coil( "Areas_ITF".A03.Safety_CtrlSafe.F_Contactor_Bloccaggio_Pareggiatore_Coda )
   END_RUNG
   RUNG wire#powerrail
      Contact( "A0302_PareggiatoreCoda".COut.PareggiatoreLong.CtrlSafe )
   END_RUNG wire#w1
   RUNG wire#powerrail
      Contact( "A03_DEBUG".Forse_Contactors_CtrlSafe )
   END_RUNG wire#w1
   RUNG wire#powerrail
      Contact( "A0302_PareggiatoreTesta".COut.Bloccaggio.CtrlSafe )
      wire#w2
      Coil( "Areas_ITF".A03.Safety_CtrlSafe.F_Contactor_Bloccaggio_Pareggiatore_Testa )
   END_RUNG
   RUNG wire#powerrail
      Contact( "A03_DEBUG".Forse_Contactors_CtrlSafe )
   END_RUNG wire#w2
   // the same network as SCL:
   "Areas_ITF".A03.Safety_CtrlSafe.F_Contactor_Bloccaggio_Pareggiatore_Coda := "A0302_PareggiatoreCoda".COut.Bloccaggio.CtrlSafe OR "A0302_PareggiatoreCoda".COut.PareggiatoreLong.CtrlSafe OR "A03_DEBUG".Forse_Contactors_CtrlSafe;
   "Areas_ITF".A03.Safety_CtrlSafe.F_Contactor_Bloccaggio_Pareggiatore_Testa := "A0302_PareggiatoreTesta".COut.Bloccaggio.CtrlSafe OR "A03_DEBUG".Forse_Contactors_CtrlSafe;
END_REGION

REGION Network 10: Ctrl Safe Area 03 HU
   // C.Olio su Centralina Cytropack
   RUNG wire#powerrail
      Contact( "A0302_HU_Cytropack".COut.CtrlSafe )
      wire#w1
      Coil( "Areas_ITF".A03.Safety_CtrlSafe.F_Contactor_HU_CYTROPAC_STO )
   END_RUNG
   RUNG wire#powerrail
      Contact( "A03_DEBUG".Forse_Contactors_CtrlSafe )
   END_RUNG wire#w1
   RUNG wire#powerrail
      Contact( "A0302_HU_Cytropack".COut.PressureRunning )
      wire#w2
      Coil( "Areas_ITF".A03.Safety_CtrlSafe.F_Contactor_HU_CYTROPAC_StandbyValve )
   END_RUNG
   RUNG wire#powerrail
      Contact( "A03_DEBUG".Forse_Contactors_CtrlSafe )
   END_RUNG wire#w2
   // the same network as SCL:
   "Areas_ITF".A03.Safety_CtrlSafe.F_Contactor_HU_CYTROPAC_STO := "A0302_HU_Cytropack".COut.CtrlSafe OR "A03_DEBUG".Forse_Contactors_CtrlSafe;
   "Areas_ITF".A03.Safety_CtrlSafe.F_Contactor_HU_CYTROPAC_StandbyValve := "A0302_HU_Cytropack".COut.PressureRunning OR "A03_DEBUG".Forse_Contactors_CtrlSafe;
END_REGION

REGION Network 12: To Area 4
   RUNG wire#powerrail
      Contact( "A0302_Manipolatore".COut.OutWorkSpace )
      Coil( "Areas_ITF".A03.ManipOutOfWorkSpace )
   END_RUNG
   RUNG wire#powerrail
      Move(in := "A0302_PareggiatoreCoda".COut.Ax, out1 => "Areas_ITF".A03.A0302_PareggiatoreCoda_COut_Ax)
   END_RUNG
   RUNG wire#powerrail
      Move(in := "A0302_PareggiatoreTesta".COut.Ax, out1 => "Areas_ITF".A03.A0302_PareggiatoreTesta_COut_Ax)
   END_RUNG
   // the same network as SCL:
   "Areas_ITF".A03.ManipOutOfWorkSpace := "A0302_Manipolatore".COut.OutWorkSpace;
   "Areas_ITF".A03.A0302_PareggiatoreCoda_COut_Ax := "A0302_PareggiatoreCoda".COut.Ax;
   "Areas_ITF".A03.A0302_PareggiatoreTesta_COut_Ax := "A0302_PareggiatoreTesta".COut.Ax;
END_REGION

REGION Network 13: To Area 2 - Richiesta PTrk su Pos1 ad Area 02
   RUNG wire#powerrail
      Contact( "A0301_Manager".COut.P1.ReqPTrk_A02 )
      Coil( "Areas_ITF".A03.A0301_Pos1_ReadyToRecive )
   END_RUNG
   // the same network as SCL:
   "Areas_ITF".A03.A0301_Pos1_ReadyToRecive := "A0301_Manager".COut.P1.ReqPTrk_A02;
END_REGION

REGION Network 14 (SCL): Area ITF Orchestrator
   // TRASFERIMENTO AREA INTERFACE SU ITF
   "Areas_ITF".A03.AreaInterface := "Area03".AreaInterface;


   "Areas_ITF".A03.Safety_SuperUser.PbSafetyReset := "A03_HMI".Area03.SuperUser.PbSafetyRst;
   "Areas_ITF".A03.Safety_SuperUser.SgnSafetyReset := "A03_HMI".Area03.SuperUser.SgnSafetyRst;

   "Areas_ITF".A03.Doors_Closed := NOT "F_DB".ZSI_Zone21.Door_NormalStop AND NOT "F_DB".ZSI_Zone23.Door_NormalStop AND NOT "F_DB".ZSI_Zone25.Door_NormalStop;
   "Areas_ITF".A03.Production_Running := "Sys".ByPass;

   //"Areas_ITF".A03.Production_Halted.Code :=;
   //"Areas_ITF".A03.Production_Halted.Message_N :=;

   "Areas_ITF".A03.SetUp_Bordatrice_Done := "A0302_Bordatrice_RegolazioneFormato".Cout.SetUp_Bordatrice_Done;

   //"MB3_Pb_Start_Ciclo_Area02" := "Areas_ITF".A02.PB.Area_DataOut_LampCycle;
   "Areas_ITF".A03.PB.MB3_Area02_PB_Start := FALSE;
   //"MB3_Pb_Start_Ciclo_Area02";
   "Areas_ITF".A03.PB.MB3_Area02_PB_Stop := FALSE;
   //"MB3_Pb_Stop_Ciclo_Area02";

   //"MB3_Pb_Start_Ciclo_Area01" := "Areas_ITF".A01.PB.Area_DataOut_LampCycle;
   "Areas_ITF".A03.PB.MB3_Area01_PB_Start := FALSE;
   //"MB3_Pb_Start_Ciclo_Area01";
   "Areas_ITF".A03.PB.MB3_Area01_PB_Stop := FALSE;
   //"MB3_Pb_Stop_Ciclo_Area01";
END_REGION
END_FUNCTION

ORGANIZATION_BLOCK "A03_OB32_CyclicInterrupt"   // OB32, LAD, CyclicInterrupt
// stored: AutoNumber false, SetENOAutomatically false
   VAR_INPUT
      Initial_Call : Bool;   // Initial call of this OB
      Event_Count : Int;   // Events discarded
   END_VAR
BEGIN

REGION Network 1
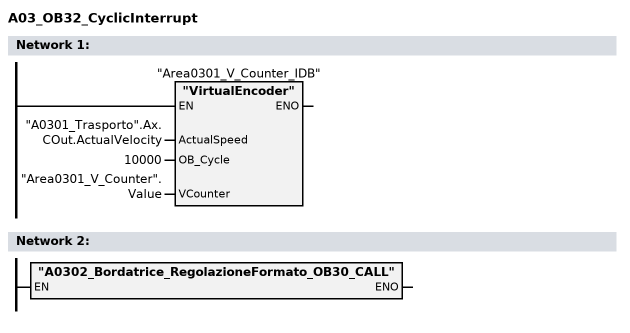
   RUNG wire#powerrail
      "Area0301_V_Counter_IDB"(ActualSpeed := "A0301_Trasporto".Ax.COut.ActualVelocity, OB_Cycle := 10000, VCounter := "Area0301_V_Counter".Value)
   END_RUNG
   // the same network as SCL:
   "Area0301_V_Counter_IDB"(ActualSpeed := "A0301_Trasporto".Ax.COut.ActualVelocity,   // "VirtualEncoder"
                           OB_Cycle := 10000,
                           VCounter := "Area0301_V_Counter".Value);
END_REGION

REGION Network 2
   RUNG wire#powerrail
      "A0302_Bordatrice_RegolazioneFormato_OB30_CALL"()
   END_RUNG
   // the same network as SCL:
   "A0302_Bordatrice_RegolazioneFormato_OB30_CALL"();
END_REGION
END_ORGANIZATION_BLOCK

FUNCTION "A03_HMI_CALL" : Void   // FC227, LAD
// stored: SetENOAutomatically false
BEGIN

REGION Network 1
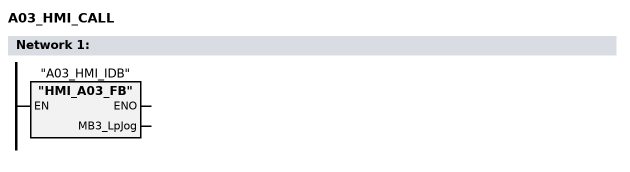
   RUNG wire#powerrail
      "A03_HMI_IDB"(MB3_LpJog =>)
   END_RUNG
   // the same network as SCL:
   "A03_HMI_IDB"();   // "HMI_A03_FB"
END_REGION
END_FUNCTION

FUNCTION_BLOCK "HMI_A03_FB"   // FB63, LAD
TITLE = HMI Managment
AUTHOR : Piemme
FAMILY : System
// stored: MemoryReserve 100, SetENOAutomatically false
   VAR_OUTPUT
      MB3_LpJog : Bool;
   END_VAR
   VAR
      MB3_Decoder { ExternalAccessible := 'False'; ExternalVisible := 'False'; ExternalWritable := 'False'} : "ButtonsHMIDecoder";
   END_VAR
   VAR CONSTANT
      "3002_TRASPORTO" : Int := 3002;
      "3011_FERMI_P1" : Int := 3011;
      "3012_FERMI_P1_SFALSATORE" : Int := 3012;
      "3021_FERMI_P2" : Int := 3021;
      "3022_FERMI_P2_SOLLEVATORE" : Int := 3022;
      "3031_FERMI_P3" : Int := 3031;
      "3032_SOLLEVA_RIBALTA" : Int := 3032;
      "3033_ROT_RIBALTA" : Int := 3033;
      "3034_ROT_RIBALTA_AX-POS" : Int := 3034;
      "3041_FERMI_P4" : Int := 3041;
      "3042_SPINTORE_LAT_VRT_P5" : Int := 3042;
      "3043_SPINTORE_LAT_ORZ_P5" : Int := 3043;
      "3044_SOLLEVATORI_P5" : Int := 3044;
      "3045_SPINTORE_LAT_OP" : Int := 3045;
      "3051_RIBALTATORE_OP-POS0" : Int := 3051;
      "3052_RIBALTATORE_OP-POS1" : Int := 3052;
      "3053_RIBALTATORE_OP-POS2" : Int := 3053;
      "3054_RIBALTATORE_OP-POS3" : Int := 3054;
      "4001_HU_CYTROPACK" : Int := 4001;
      "4011_SPINTORE_OP" : Int := 4011;
      "4012_SPINTORE_AX" : Int := 4012;
      "4013_SPINTORE_VRT" : Int := 4013;
      "4014_SPINTORE_ORZ" : Int := 4014;
      "4021_BORDATRICE_AX" : Int := 4021;
      "4031_RULLIERA_OP" : Int := 4031;
      "4032_RULLIERA_AX" : Int := 4032;
      "4033_BORDATRICE_REG-CASSETTA" : Int := 4033;
      "4034_BORDATRICE_PASS01" : Int := 4034;
      "4035_BORDATRICE_PASS02" : Int := 4035;
      "4036_BORDATRICE_PASS03" : Int := 4036;
      "4037_BORDATRICE_PASS04" : Int := 4037;
      "4038_BORDATRICE_REG-CASSETTA_AX-POS" : Int := 4038;
      "4041_CENTRATORI_OP" : Int := 4041;
      "4042_CENTRATORI_CENTRAGGIO" : Int := 4042;
      "4043_CENTRATORI_SOLLEVAMENTO" : Int := 4043;
      "4051_PAREGGIATORE_CODA_OP" : Int := 4051;
      "4052_PAREGGIATORE_CODA_AX" : Int := 4052;
      "4053_PAREGGIATORE_CODA_BLOCCAGGIO" : Int := 4053;
      "4054_PAREGGIATORE_CODA_BATTUTAVERTICALE" : Int := 4054;
      "4055_PAREGGIATORE_CODA_PAREGGIATORELONGIT" : Int := 4055;
      "4061_PAREGGIATORE_TESTA_OP" : Int := 4061;
      "4062_PAREGGIATORE_TESTA_AX" : Int := 4062;
      "4063_PAREGGIATORE_TESTA_BLOCCAGGIO" : Int := 4063;
      "4064_PAREGGIATORE_TESTA_SOLLEVAMENTO" : Int := 4064;
      "4065_PAREGGIATORE_TESTA_CENTRAGGIO" : Int := 4065;
      "4066_PAREGG_TESTA_AX_POS" : Int := 4066;
      "4067_PAREGG_CODA_AX_POS" : Int := 4067;
      "4070_MANIPOLATORE_OP" : Int := 4070;
      "4071_MANIPOLATORE_AX" : Int := 4071;
      "4072_MANIPOLATORE_AX-POS" : Int := 4072;
      "4073_MANIPOLATORE_MAGNETE" : Int := 4073;
      "4074_MANIPOLATORE_SOLLEVATORE" : Int := 4074;
      "4080_BORDATRICE_PASS01_LATO-OP" : Int := 4080;
      "4081_BORDATRICE_PASS01_LATO-MOT" : Int := 4081;
      "4082_BORDATRICE_PASS02_LATO-OP" : Int := 4082;
      "4083_BORDATRICE_PASS02_LATO-MOT" : Int := 4083;
      "4084_BORDATRICE_PASS03_LATO-OP" : Int := 4084;
      "4085_BORDATRICE_PASS03_LATO-MOT" : Int := 4085;
      "4086_BORDATRICE_PASS04_LATO-OP" : Int := 4086;
      "4087_BORDATRICE_PASS04_LATO-MOT" : Int := 4087;
      "4088_BORDATRICE_PASS01-COMBO_AX-POS" : Int := 4088;
      "4089_BORDATRICE_PASS02-COMBO_AX-POS" : Int := 4089;
      "4090_BORDATRICE_PASS03-COMBO_AX-POS" : Int := 4090;
      "4091_BORDATRICE_PASS04-COMBO_AX-POS" : Int := 4091;
      "4092_BORDATRICE_PASS01-LATO-OP_AX-POS" : Int := 4092;
      "4093_BORDATRICE_PASS01-LATO-MOT_AX-POS" : Int := 4093;
      "4094_BORDATRICE_PASS02-LATO-OP_AX-POS" : Int := 4094;
      "4095_BORDATRICE_PASS02-LATO-MOT_AX-POS" : Int := 4095;
      "4096_BORDATRICE_PASS03-LATO-OP_AX-POS" : Int := 4096;
      "4097_BORDATRICE_PASS03-LATO-MOT_AX-POS" : Int := 4097;
      "4098_BORDATRICE_PASS04-LATO-OP_AX-POS" : Int := 4098;
      "4099_BORDATRICE_PASS04-LATO-MOT_AX-POS" : Int := 4099;
      "5001_SPALLA_OP_POS" : Int := 5001;
      "5002_SPALLA_TESTA_AX_JOG" : Int := 5002;
      "5003_SPALLA_TESTA_AX_POS" : Int := 5003;
      "5005_SPALLA_CODA_AX" : Int := 5005;
      "5006_SPALLA_CODA_AX_POS" : Int := 5006;
      "5011_SPINTORE_OP" : Int := 5011;
      "5012_SPINTORE_VRT" : Int := 5012;
      "5013_SPINTORE_ORZ" : Int := 5013;
      "5021_TRASLAZIONE_OP_VAI_A_PRELIEVO" : Int := 5021;
      "5022_TRASLAZIONE_OP_PRELIEVO" : Int := 5022;
      "5023_TRASLAZIONE_OP_VAI_A_DEPOSITO" : Int := 5023;
      "5024_TRASLAZIONE_OP_DEPOSITO" : Int := 5024;
      "5025_TRASLAZIONE_AX_JOG" : Int := 5025;
      "5026_TRASLAZIONE_AX_POS" : Int := 5026;
      "5027_TRASLAZIONE_MANIP_SOSTEGNO" : Int := 5027;
      "5028_TRASLAZIONE_MANIP_PAREGGIATORE" : Int := 5028;
      "5029_TRASLAZIONE_SOSTEGNO_VERTICALE" : Int := 5029;
      "5031_SOLLEVAMENTO_OP" : Int := 5031;
      "5032_SOLLEVAMENTO_AX_JOG" : Int := 5032;
      "5033_SOLLEVAMENTO_AX_POS" : Int := 5033;
      "5041_PALETTIANTIRIBALTAMENTO_OP" : Int := 5041;
      "5042_PALETTIANTIRIBALTAMENTO_TESTA_POS0" : Int := 5042;
      "5043_PALETTIANTIRIBALTAMENTO_TESTA_POS1" : Int := 5043;
      "5044_PALETTIANTIRIBALTAMENTO_TESTA_POS2" : Int := 5044;
      "5046_PALETTIANTIRIBALTAMENTO_CODA_POS0" : Int := 5046;
      "5047_PALETTIANTIRIBALTAMENTO_CODA_POS1" : Int := 5047;
      "5048_PALETTIANTIRIBALTAMENTO_CODA_POS2" : Int := 5048;
      "5051_SOSTEGNO_TESTA_AX_JOG" : Int := 5051;
      "5052_SOSTEGNO_TESTA_AX_POS" : Int := 5052;
      "5053_SOSTEGNO_CODA_AX_JOG" : Int := 5053;
      "5054_SOSTEGNO_CODA_AX_POS" : Int := 5054;
      "6001_NAVETTA_OP_VAI_A_PRELIEVO" : Int := 6001;
      "6002_NAVETTA_OP_PRELIEVO" : Int := 6002;
      "6003_NAVETTA_OP_VAI_A_DEPOSITO" : Int := 6003;
      "6004_NAVETTA_OP_DEPOSITO" : Int := 6004;
      "6005_NAVETTA_AX" : Int := 6005;
      "6006_NAVETTA_PALETTI_INTERNI" : Int := 6006;
      "6007_NAVETTA_PALETTI_ESTERNI" : Int := 6007;
   END_VAR
   VAR_TEMP   // added for the SCL form of the ladder/FBD networks
      _w1 : Bool;
   END_VAR
BEGIN

REGION Network 2: <<< MB3 MANUALS OPERATIONS >>>
END_REGION

REGION Network 3 (SCL): Reset Op
   #MB3_Decoder.OpEnabled := FALSE;
   #MB3_Decoder.OpRunning := FALSE;
   #MB3_Decoder.OpDone := FALSE;
END_REGION

REGION Network 4: <<<<<<<<< A0301 STAZIONE 1 >>>>>>>>>>>>>
END_REGION

REGION Network 5: MB3 Code 3002 - Trasporto
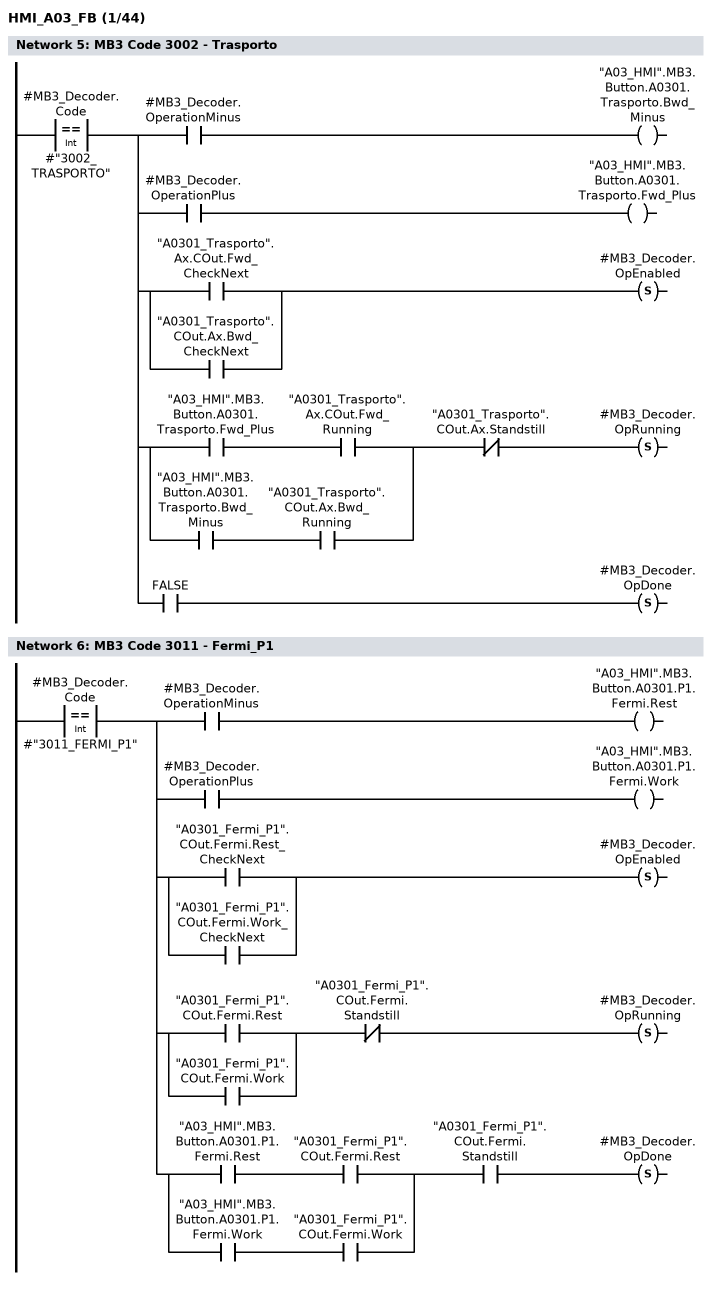
   RUNG wire#powerrail
      { S7_Templates := "SrcType := Int" } EQ_Contact(in1 := #MB3_Decoder.Code, in2 := #"3002_TRASPORTO")
      wire#w1
      Contact( #MB3_Decoder.OperationMinus )
      Coil( "A03_HMI".MB3.Button.A0301.Trasporto.Bwd_Minus )
   END_RUNG
   RUNG wire#w1
      Contact( #MB3_Decoder.OperationPlus )
      Coil( "A03_HMI".MB3.Button.A0301.Trasporto.Fwd_Plus )
   END_RUNG
   RUNG wire#w1
      Contact( "A0301_Trasporto".Ax.COut.Fwd_CheckNext )
      wire#w2
      S_Coil( #MB3_Decoder.OpEnabled )
   END_RUNG
   RUNG wire#w1
      Contact( "A0301_Trasporto".COut.Ax.Bwd_CheckNext )
   END_RUNG wire#w2
   RUNG wire#w1
      Contact( "A03_HMI".MB3.Button.A0301.Trasporto.Fwd_Plus )
      Contact( "A0301_Trasporto".Ax.COut.Fwd_Running )
      wire#w3
      I_Contact( "A0301_Trasporto".COut.Ax.Standstill )
      S_Coil( #MB3_Decoder.OpRunning )
   END_RUNG
   RUNG wire#w1
      Contact( "A03_HMI".MB3.Button.A0301.Trasporto.Bwd_Minus )
      Contact( "A0301_Trasporto".COut.Ax.Bwd_Running )
   END_RUNG wire#w3
   RUNG wire#w1
      Contact( FALSE )
      S_Coil( #MB3_Decoder.OpDone )
   END_RUNG
   // the same network as SCL:
   #_w1 := #MB3_Decoder.Code = #"3002_TRASPORTO";
   "A03_HMI".MB3.Button.A0301.Trasporto.Bwd_Minus := #_w1 AND #MB3_Decoder.OperationMinus;
   "A03_HMI".MB3.Button.A0301.Trasporto.Fwd_Plus := #_w1 AND #MB3_Decoder.OperationPlus;
   IF #_w1 AND ("A0301_Trasporto".Ax.COut.Fwd_CheckNext OR "A0301_Trasporto".COut.Ax.Bwd_CheckNext) THEN
       #MB3_Decoder.OpEnabled := TRUE;
   END_IF;
   IF #_w1 AND (("A03_HMI".MB3.Button.A0301.Trasporto.Fwd_Plus AND "A0301_Trasporto".Ax.COut.Fwd_Running) OR ("A03_HMI".MB3.Button.A0301.Trasporto.Bwd_Minus AND "A0301_Trasporto".COut.Ax.Bwd_Running)) AND NOT "A0301_Trasporto".COut.Ax.Standstill THEN
       #MB3_Decoder.OpRunning := TRUE;
   END_IF;
   IF #_w1 AND FALSE THEN #MB3_Decoder.OpDone := TRUE; END_IF;
END_REGION

REGION Network 6: MB3 Code 3011 - Fermi_P1
   RUNG wire#powerrail
      { S7_Templates := "SrcType := Int" } EQ_Contact(in1 := #MB3_Decoder.Code, in2 := #"3011_FERMI_P1")
      wire#w1
      Contact( #MB3_Decoder.OperationMinus )
      Coil( "A03_HMI".MB3.Button.A0301.P1.Fermi.Rest )
   END_RUNG
   RUNG wire#w1
      Contact( #MB3_Decoder.OperationPlus )
      Coil( "A03_HMI".MB3.Button.A0301.P1.Fermi.Work )
   END_RUNG
   RUNG wire#w1
      Contact( "A0301_Fermi_P1".COut.Fermi.Rest_CheckNext )
      wire#w2
      S_Coil( #MB3_Decoder.OpEnabled )
   END_RUNG
   RUNG wire#w1
      Contact( "A0301_Fermi_P1".COut.Fermi.Work_CheckNext )
   END_RUNG wire#w2
   RUNG wire#w1
      Contact( "A0301_Fermi_P1".COut.Fermi.Rest )
      wire#w3
      I_Contact( "A0301_Fermi_P1".COut.Fermi.Standstill )
      S_Coil( #MB3_Decoder.OpRunning )
   END_RUNG
   RUNG wire#w1
      Contact( "A0301_Fermi_P1".COut.Fermi.Work )
   END_RUNG wire#w3
   RUNG wire#w1
      Contact( "A03_HMI".MB3.Button.A0301.P1.Fermi.Rest )
      Contact( "A0301_Fermi_P1".COut.Fermi.Rest )
      wire#w4
      Contact( "A0301_Fermi_P1".COut.Fermi.Standstill )
      S_Coil( #MB3_Decoder.OpDone )
   END_RUNG
   RUNG wire#w1
      Contact( "A03_HMI".MB3.Button.A0301.P1.Fermi.Work )
      Contact( "A0301_Fermi_P1".COut.Fermi.Work )
   END_RUNG wire#w4
   // the same network as SCL:
   #_w1 := #MB3_Decoder.Code = #"3011_FERMI_P1";
   "A03_HMI".MB3.Button.A0301.P1.Fermi.Rest := #_w1 AND #MB3_Decoder.OperationMinus;
   "A03_HMI".MB3.Button.A0301.P1.Fermi.Work := #_w1 AND #MB3_Decoder.OperationPlus;
   IF #_w1 AND ("A0301_Fermi_P1".COut.Fermi.Rest_CheckNext OR "A0301_Fermi_P1".COut.Fermi.Work_CheckNext) THEN
       #MB3_Decoder.OpEnabled := TRUE;
   END_IF;
   IF #_w1 AND ("A0301_Fermi_P1".COut.Fermi.Rest OR "A0301_Fermi_P1".COut.Fermi.Work) AND NOT "A0301_Fermi_P1".COut.Fermi.Standstill THEN
       #MB3_Decoder.OpRunning := TRUE;
   END_IF;
   IF #_w1 AND (("A03_HMI".MB3.Button.A0301.P1.Fermi.Rest AND "A0301_Fermi_P1".COut.Fermi.Rest) OR ("A03_HMI".MB3.Button.A0301.P1.Fermi.Work AND "A0301_Fermi_P1".COut.Fermi.Work)) AND "A0301_Fermi_P1".COut.Fermi.Standstill THEN
       #MB3_Decoder.OpDone := TRUE;
   END_IF;
END_REGION

REGION Network 7: MB3 Code 3012 - P1 Sfalsatore
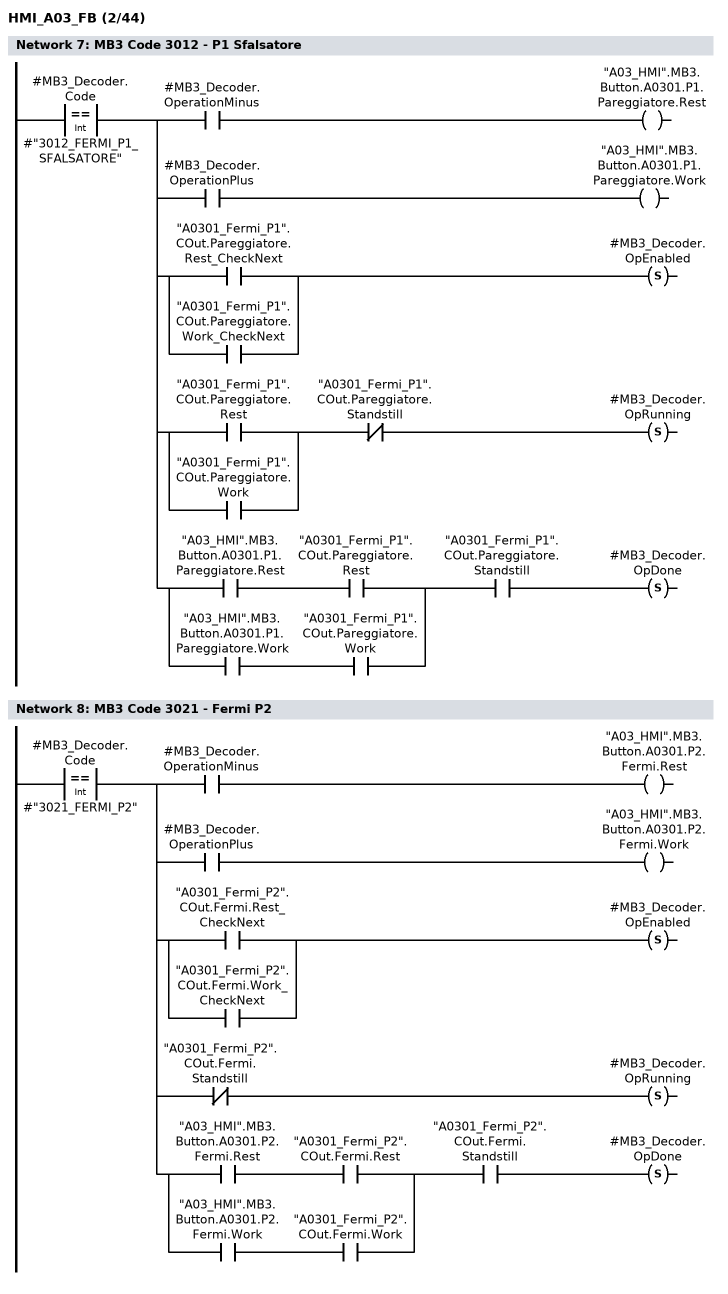
   RUNG wire#powerrail
      { S7_Templates := "SrcType := Int" } EQ_Contact(in1 := #MB3_Decoder.Code, in2 := #"3012_FERMI_P1_SFALSATORE")
      wire#w1
      Contact( #MB3_Decoder.OperationMinus )
      Coil( "A03_HMI".MB3.Button.A0301.P1.Pareggiatore.Rest )
   END_RUNG
   RUNG wire#w1
      Contact( #MB3_Decoder.OperationPlus )
      Coil( "A03_HMI".MB3.Button.A0301.P1.Pareggiatore.Work )
   END_RUNG
   RUNG wire#w1
      Contact( "A0301_Fermi_P1".COut.Pareggiatore.Rest_CheckNext )
      wire#w2
      S_Coil( #MB3_Decoder.OpEnabled )
   END_RUNG
   RUNG wire#w1
      Contact( "A0301_Fermi_P1".COut.Pareggiatore.Work_CheckNext )
   END_RUNG wire#w2
   RUNG wire#w1
      Contact( "A0301_Fermi_P1".COut.Pareggiatore.Rest )
      wire#w3
      I_Contact( "A0301_Fermi_P1".COut.Pareggiatore.Standstill )
      S_Coil( #MB3_Decoder.OpRunning )
   END_RUNG
   RUNG wire#w1
      Contact( "A0301_Fermi_P1".COut.Pareggiatore.Work )
   END_RUNG wire#w3
   RUNG wire#w1
      Contact( "A03_HMI".MB3.Button.A0301.P1.Pareggiatore.Rest )
      Contact( "A0301_Fermi_P1".COut.Pareggiatore.Rest )
      wire#w4
      Contact( "A0301_Fermi_P1".COut.Pareggiatore.Standstill )
      S_Coil( #MB3_Decoder.OpDone )
   END_RUNG
   RUNG wire#w1
      Contact( "A03_HMI".MB3.Button.A0301.P1.Pareggiatore.Work )
      Contact( "A0301_Fermi_P1".COut.Pareggiatore.Work )
   END_RUNG wire#w4
   // the same network as SCL:
   #_w1 := #MB3_Decoder.Code = #"3012_FERMI_P1_SFALSATORE";
   "A03_HMI".MB3.Button.A0301.P1.Pareggiatore.Rest := #_w1 AND #MB3_Decoder.OperationMinus;
   "A03_HMI".MB3.Button.A0301.P1.Pareggiatore.Work := #_w1 AND #MB3_Decoder.OperationPlus;
   IF #_w1 AND ("A0301_Fermi_P1".COut.Pareggiatore.Rest_CheckNext OR "A0301_Fermi_P1".COut.Pareggiatore.Work_CheckNext) THEN
       #MB3_Decoder.OpEnabled := TRUE;
   END_IF;
   IF #_w1 AND ("A0301_Fermi_P1".COut.Pareggiatore.Rest OR "A0301_Fermi_P1".COut.Pareggiatore.Work) AND NOT "A0301_Fermi_P1".COut.Pareggiatore.Standstill THEN
       #MB3_Decoder.OpRunning := TRUE;
   END_IF;
   IF #_w1 AND (("A03_HMI".MB3.Button.A0301.P1.Pareggiatore.Rest AND "A0301_Fermi_P1".COut.Pareggiatore.Rest) OR ("A03_HMI".MB3.Button.A0301.P1.Pareggiatore.Work AND "A0301_Fermi_P1".COut.Pareggiatore.Work)) AND "A0301_Fermi_P1".COut.Pareggiatore.Standstill THEN
       #MB3_Decoder.OpDone := TRUE;
   END_IF;
END_REGION

REGION Network 8: MB3 Code 3021 - Fermi P2
   RUNG wire#powerrail
      { S7_Templates := "SrcType := Int" } EQ_Contact(in1 := #MB3_Decoder.Code, in2 := #"3021_FERMI_P2")
      wire#w1
      Contact( #MB3_Decoder.OperationMinus )
      Coil( "A03_HMI".MB3.Button.A0301.P2.Fermi.Rest )
   END_RUNG
   RUNG wire#w1
      Contact( #MB3_Decoder.OperationPlus )
      Coil( "A03_HMI".MB3.Button.A0301.P2.Fermi.Work )
   END_RUNG
   RUNG wire#w1
      Contact( "A0301_Fermi_P2".COut.Fermi.Rest_CheckNext )
      wire#w2
      S_Coil( #MB3_Decoder.OpEnabled )
   END_RUNG
   RUNG wire#w1
      Contact( "A0301_Fermi_P2".COut.Fermi.Work_CheckNext )
   END_RUNG wire#w2
   RUNG wire#w1
      I_Contact( "A0301_Fermi_P2".COut.Fermi.Standstill )
      S_Coil( #MB3_Decoder.OpRunning )
   END_RUNG
   RUNG wire#w1
      Contact( "A03_HMI".MB3.Button.A0301.P2.Fermi.Rest )
      Contact( "A0301_Fermi_P2".COut.Fermi.Rest )
      wire#w3
      Contact( "A0301_Fermi_P2".COut.Fermi.Standstill )
      S_Coil( #MB3_Decoder.OpDone )
   END_RUNG
   RUNG wire#w1
      Contact( "A03_HMI".MB3.Button.A0301.P2.Fermi.Work )
      Contact( "A0301_Fermi_P2".COut.Fermi.Work )
   END_RUNG wire#w3
   // the same network as SCL:
   #_w1 := #MB3_Decoder.Code = #"3021_FERMI_P2";
   "A03_HMI".MB3.Button.A0301.P2.Fermi.Rest := #_w1 AND #MB3_Decoder.OperationMinus;
   "A03_HMI".MB3.Button.A0301.P2.Fermi.Work := #_w1 AND #MB3_Decoder.OperationPlus;
   IF #_w1 AND ("A0301_Fermi_P2".COut.Fermi.Rest_CheckNext OR "A0301_Fermi_P2".COut.Fermi.Work_CheckNext) THEN
       #MB3_Decoder.OpEnabled := TRUE;
   END_IF;
   IF #_w1 AND NOT "A0301_Fermi_P2".COut.Fermi.Standstill THEN #MB3_Decoder.OpRunning := TRUE; END_IF;
   IF #_w1 AND (("A03_HMI".MB3.Button.A0301.P2.Fermi.Rest AND "A0301_Fermi_P2".COut.Fermi.Rest) OR ("A03_HMI".MB3.Button.A0301.P2.Fermi.Work AND "A0301_Fermi_P2".COut.Fermi.Work)) AND "A0301_Fermi_P2".COut.Fermi.Standstill THEN
       #MB3_Decoder.OpDone := TRUE;
   END_IF;
END_REGION

REGION Network 9: MB3 Code 3022 - P2 - Sollevatore
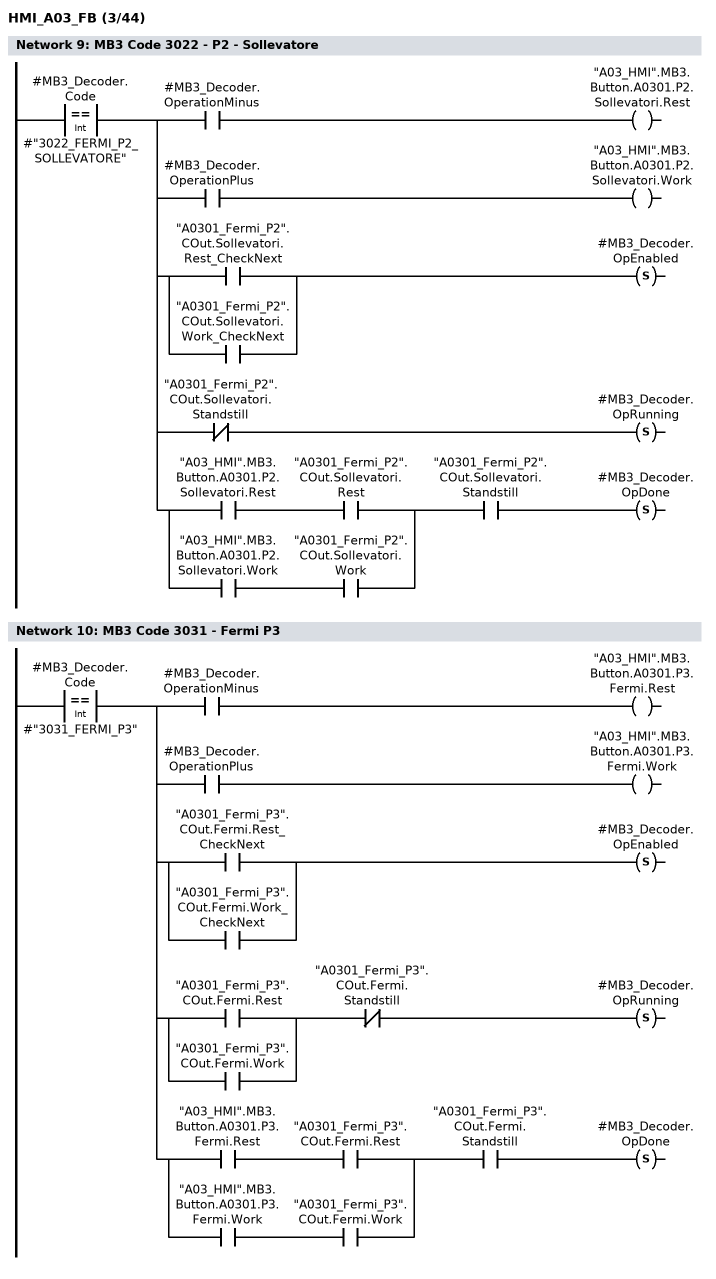
   RUNG wire#powerrail
      { S7_Templates := "SrcType := Int" } EQ_Contact(in1 := #MB3_Decoder.Code, in2 := #"3022_FERMI_P2_SOLLEVATORE")
      wire#w1
      Contact( #MB3_Decoder.OperationMinus )
      Coil( "A03_HMI".MB3.Button.A0301.P2.Sollevatori.Rest )
   END_RUNG
   RUNG wire#w1
      Contact( #MB3_Decoder.OperationPlus )
      Coil( "A03_HMI".MB3.Button.A0301.P2.Sollevatori.Work )
   END_RUNG
   RUNG wire#w1
      Contact( "A0301_Fermi_P2".COut.Sollevatori.Rest_CheckNext )
      wire#w2
      S_Coil( #MB3_Decoder.OpEnabled )
   END_RUNG
   RUNG wire#w1
      Contact( "A0301_Fermi_P2".COut.Sollevatori.Work_CheckNext )
   END_RUNG wire#w2
   RUNG wire#w1
      I_Contact( "A0301_Fermi_P2".COut.Sollevatori.Standstill )
      S_Coil( #MB3_Decoder.OpRunning )
   END_RUNG
   RUNG wire#w1
      Contact( "A03_HMI".MB3.Button.A0301.P2.Sollevatori.Rest )
      Contact( "A0301_Fermi_P2".COut.Sollevatori.Rest )
      wire#w3
      Contact( "A0301_Fermi_P2".COut.Sollevatori.Standstill )
      S_Coil( #MB3_Decoder.OpDone )
   END_RUNG
   RUNG wire#w1
      Contact( "A03_HMI".MB3.Button.A0301.P2.Sollevatori.Work )
      Contact( "A0301_Fermi_P2".COut.Sollevatori.Work )
   END_RUNG wire#w3
   // the same network as SCL:
   #_w1 := #MB3_Decoder.Code = #"3022_FERMI_P2_SOLLEVATORE";
   "A03_HMI".MB3.Button.A0301.P2.Sollevatori.Rest := #_w1 AND #MB3_Decoder.OperationMinus;
   "A03_HMI".MB3.Button.A0301.P2.Sollevatori.Work := #_w1 AND #MB3_Decoder.OperationPlus;
   IF #_w1 AND ("A0301_Fermi_P2".COut.Sollevatori.Rest_CheckNext OR "A0301_Fermi_P2".COut.Sollevatori.Work_CheckNext) THEN
       #MB3_Decoder.OpEnabled := TRUE;
   END_IF;
   IF #_w1 AND NOT "A0301_Fermi_P2".COut.Sollevatori.Standstill THEN #MB3_Decoder.OpRunning := TRUE; END_IF;
   IF #_w1 AND (("A03_HMI".MB3.Button.A0301.P2.Sollevatori.Rest AND "A0301_Fermi_P2".COut.Sollevatori.Rest) OR ("A03_HMI".MB3.Button.A0301.P2.Sollevatori.Work AND "A0301_Fermi_P2".COut.Sollevatori.Work)) AND "A0301_Fermi_P2".COut.Sollevatori.Standstill THEN
       #MB3_Decoder.OpDone := TRUE;
   END_IF;
END_REGION

REGION Network 10: MB3 Code 3031 - Fermi P3
   RUNG wire#powerrail
      { S7_Templates := "SrcType := Int" } EQ_Contact(in1 := #MB3_Decoder.Code, in2 := #"3031_FERMI_P3")
      wire#w1
      Contact( #MB3_Decoder.OperationMinus )
      Coil( "A03_HMI".MB3.Button.A0301.P3.Fermi.Rest )
   END_RUNG
   RUNG wire#w1
      Contact( #MB3_Decoder.OperationPlus )
      Coil( "A03_HMI".MB3.Button.A0301.P3.Fermi.Work )
   END_RUNG
   RUNG wire#w1
      Contact( "A0301_Fermi_P3".COut.Fermi.Rest_CheckNext )
      wire#w2
      S_Coil( #MB3_Decoder.OpEnabled )
   END_RUNG
   RUNG wire#w1
      Contact( "A0301_Fermi_P3".COut.Fermi.Work_CheckNext )
   END_RUNG wire#w2
   RUNG wire#w1
      Contact( "A0301_Fermi_P3".COut.Fermi.Rest )
      wire#w3
      I_Contact( "A0301_Fermi_P3".COut.Fermi.Standstill )
      S_Coil( #MB3_Decoder.OpRunning )
   END_RUNG
   RUNG wire#w1
      Contact( "A0301_Fermi_P3".COut.Fermi.Work )
   END_RUNG wire#w3
   RUNG wire#w1
      Contact( "A03_HMI".MB3.Button.A0301.P3.Fermi.Rest )
      Contact( "A0301_Fermi_P3".COut.Fermi.Rest )
      wire#w4
      Contact( "A0301_Fermi_P3".COut.Fermi.Standstill )
      S_Coil( #MB3_Decoder.OpDone )
   END_RUNG
   RUNG wire#w1
      Contact( "A03_HMI".MB3.Button.A0301.P3.Fermi.Work )
      Contact( "A0301_Fermi_P3".COut.Fermi.Work )
   END_RUNG wire#w4
   // the same network as SCL:
   #_w1 := #MB3_Decoder.Code = #"3031_FERMI_P3";
   "A03_HMI".MB3.Button.A0301.P3.Fermi.Rest := #_w1 AND #MB3_Decoder.OperationMinus;
   "A03_HMI".MB3.Button.A0301.P3.Fermi.Work := #_w1 AND #MB3_Decoder.OperationPlus;
   IF #_w1 AND ("A0301_Fermi_P3".COut.Fermi.Rest_CheckNext OR "A0301_Fermi_P3".COut.Fermi.Work_CheckNext) THEN
       #MB3_Decoder.OpEnabled := TRUE;
   END_IF;
   IF #_w1 AND ("A0301_Fermi_P3".COut.Fermi.Rest OR "A0301_Fermi_P3".COut.Fermi.Work) AND NOT "A0301_Fermi_P3".COut.Fermi.Standstill THEN
       #MB3_Decoder.OpRunning := TRUE;
   END_IF;
   IF #_w1 AND (("A03_HMI".MB3.Button.A0301.P3.Fermi.Rest AND "A0301_Fermi_P3".COut.Fermi.Rest) OR ("A03_HMI".MB3.Button.A0301.P3.Fermi.Work AND "A0301_Fermi_P3".COut.Fermi.Work)) AND "A0301_Fermi_P3".COut.Fermi.Standstill THEN
       #MB3_Decoder.OpDone := TRUE;
   END_IF;
END_REGION

REGION Network 11: MB3 Code 3032 - Solleva Ribalta
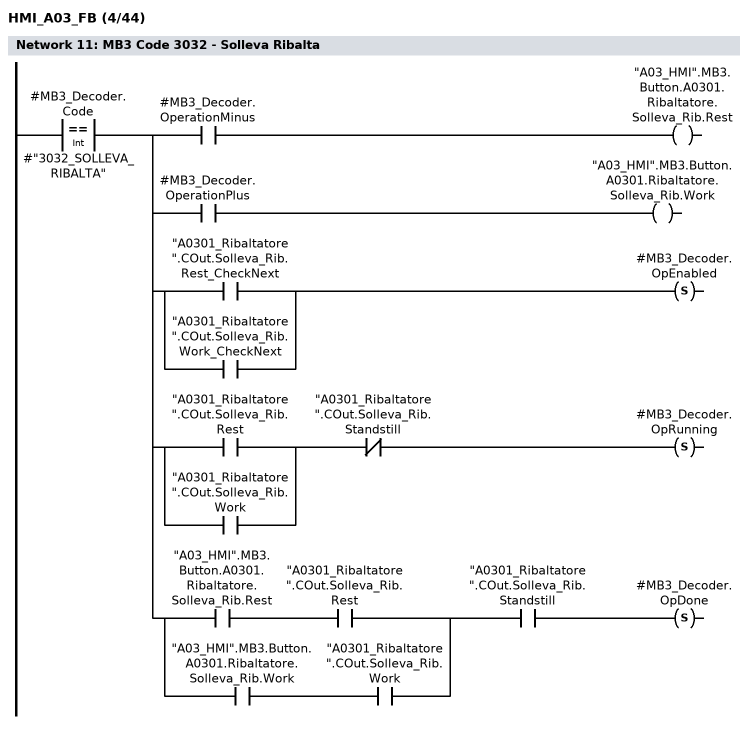
   RUNG wire#powerrail
      { S7_Templates := "SrcType := Int" } EQ_Contact(in1 := #MB3_Decoder.Code, in2 := #"3032_SOLLEVA_RIBALTA")
      wire#w1
      Contact( #MB3_Decoder.OperationMinus )
      Coil( "A03_HMI".MB3.Button.A0301.Ribaltatore.Solleva_Rib.Rest )
   END_RUNG
   RUNG wire#w1
      Contact( #MB3_Decoder.OperationPlus )
      Coil( "A03_HMI".MB3.Button.A0301.Ribaltatore.Solleva_Rib.Work )
   END_RUNG
   RUNG wire#w1
      Contact( "A0301_Ribaltatore".COut.Solleva_Rib.Rest_CheckNext )
      wire#w2
      S_Coil( #MB3_Decoder.OpEnabled )
   END_RUNG
   RUNG wire#w1
      Contact( "A0301_Ribaltatore".COut.Solleva_Rib.Work_CheckNext )
   END_RUNG wire#w2
   RUNG wire#w1
      Contact( "A0301_Ribaltatore".COut.Solleva_Rib.Rest )
      wire#w3
      I_Contact( "A0301_Ribaltatore".COut.Solleva_Rib.Standstill )
      S_Coil( #MB3_Decoder.OpRunning )
   END_RUNG
   RUNG wire#w1
      Contact( "A0301_Ribaltatore".COut.Solleva_Rib.Work )
   END_RUNG wire#w3
   RUNG wire#w1
      Contact( "A03_HMI".MB3.Button.A0301.Ribaltatore.Solleva_Rib.Rest )
      Contact( "A0301_Ribaltatore".COut.Solleva_Rib.Rest )
      wire#w4
      Contact( "A0301_Ribaltatore".COut.Solleva_Rib.Standstill )
      S_Coil( #MB3_Decoder.OpDone )
   END_RUNG
   RUNG wire#w1
      Contact( "A03_HMI".MB3.Button.A0301.Ribaltatore.Solleva_Rib.Work )
      Contact( "A0301_Ribaltatore".COut.Solleva_Rib.Work )
   END_RUNG wire#w4
   // the same network as SCL:
   #_w1 := #MB3_Decoder.Code = #"3032_SOLLEVA_RIBALTA";
   "A03_HMI".MB3.Button.A0301.Ribaltatore.Solleva_Rib.Rest := #_w1 AND #MB3_Decoder.OperationMinus;
   "A03_HMI".MB3.Button.A0301.Ribaltatore.Solleva_Rib.Work := #_w1 AND #MB3_Decoder.OperationPlus;
   IF #_w1 AND ("A0301_Ribaltatore".COut.Solleva_Rib.Rest_CheckNext OR "A0301_Ribaltatore".COut.Solleva_Rib.Work_CheckNext) THEN
       #MB3_Decoder.OpEnabled := TRUE;
   END_IF;
   IF #_w1 AND ("A0301_Ribaltatore".COut.Solleva_Rib.Rest OR "A0301_Ribaltatore".COut.Solleva_Rib.Work) AND NOT "A0301_Ribaltatore".COut.Solleva_Rib.Standstill THEN
       #MB3_Decoder.OpRunning := TRUE;
   END_IF;
   IF #_w1 AND (("A03_HMI".MB3.Button.A0301.Ribaltatore.Solleva_Rib.Rest AND "A0301_Ribaltatore".COut.Solleva_Rib.Rest) OR ("A03_HMI".MB3.Button.A0301.Ribaltatore.Solleva_Rib.Work AND "A0301_Ribaltatore".COut.Solleva_Rib.Work)) AND "A0301_Ribaltatore".COut.Solleva_Rib.Standstill THEN
       #MB3_Decoder.OpDone := TRUE;
   END_IF;
END_REGION

REGION Network 12: MB3 Code 3033 - Rotazione Ribalta
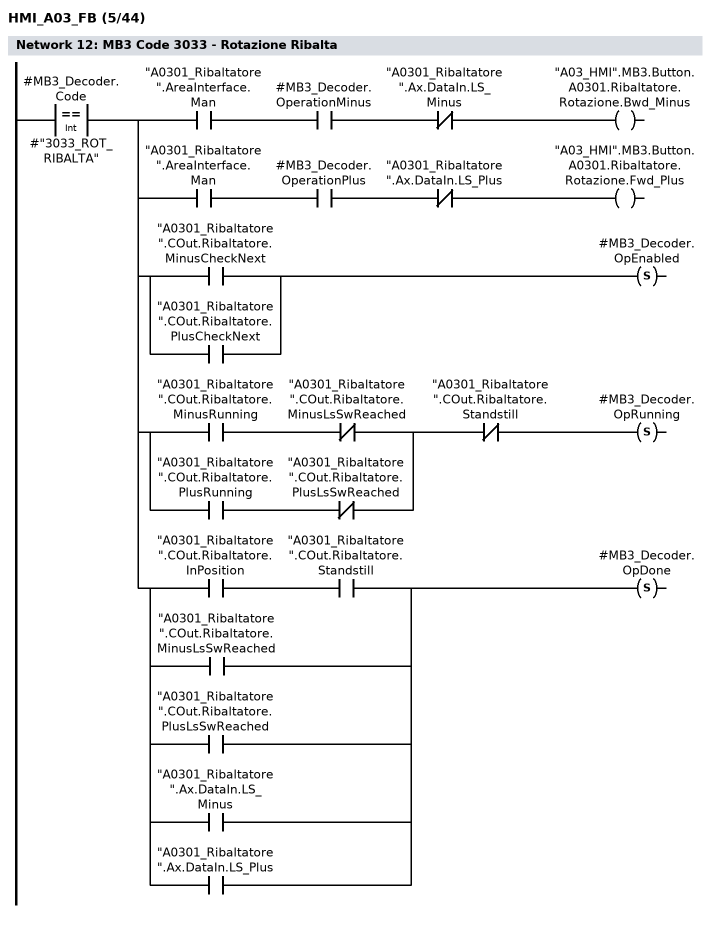
   RUNG wire#powerrail
      { S7_Templates := "SrcType := Int" } EQ_Contact(in1 := #MB3_Decoder.Code, in2 := #"3033_ROT_RIBALTA")
      wire#w1
      Contact( "A0301_Ribaltatore".AreaInterface.Man )
      Contact( #MB3_Decoder.OperationMinus )
      I_Contact( "A0301_Ribaltatore".Ax.DataIn.LS_Minus )
      Coil( "A03_HMI".MB3.Button.A0301.Ribaltatore.Rotazione.Bwd_Minus )
   END_RUNG
   RUNG wire#w1
      Contact( "A0301_Ribaltatore".AreaInterface.Man )
      Contact( #MB3_Decoder.OperationPlus )
      I_Contact( "A0301_Ribaltatore".Ax.DataIn.LS_Plus )
      Coil( "A03_HMI".MB3.Button.A0301.Ribaltatore.Rotazione.Fwd_Plus )
   END_RUNG
   RUNG wire#w1
      Contact( "A0301_Ribaltatore".COut.Ribaltatore.MinusCheckNext )
      wire#w2
      S_Coil( #MB3_Decoder.OpEnabled )
   END_RUNG
   RUNG wire#w1
      Contact( "A0301_Ribaltatore".COut.Ribaltatore.PlusCheckNext )
   END_RUNG wire#w2
   RUNG wire#w1
      Contact( "A0301_Ribaltatore".COut.Ribaltatore.MinusRunning )
      I_Contact( "A0301_Ribaltatore".COut.Ribaltatore.MinusLsSwReached )
      wire#w3
      I_Contact( "A0301_Ribaltatore".COut.Ribaltatore.Standstill )
      S_Coil( #MB3_Decoder.OpRunning )
   END_RUNG
   RUNG wire#w1
      Contact( "A0301_Ribaltatore".COut.Ribaltatore.PlusRunning )
      I_Contact( "A0301_Ribaltatore".COut.Ribaltatore.PlusLsSwReached )
   END_RUNG wire#w3
   RUNG wire#w1
      Contact( "A0301_Ribaltatore".COut.Ribaltatore.InPosition )
      Contact( "A0301_Ribaltatore".COut.Ribaltatore.Standstill )
      wire#w4
      S_Coil( #MB3_Decoder.OpDone )
   END_RUNG
   RUNG wire#w1
      Contact( "A0301_Ribaltatore".COut.Ribaltatore.MinusLsSwReached )
   END_RUNG wire#w4
   RUNG wire#w1
      Contact( "A0301_Ribaltatore".COut.Ribaltatore.PlusLsSwReached )
   END_RUNG wire#w4
   RUNG wire#w1
      Contact( "A0301_Ribaltatore".Ax.DataIn.LS_Minus )
   END_RUNG wire#w4
   RUNG wire#w1
      Contact( "A0301_Ribaltatore".Ax.DataIn.LS_Plus )
   END_RUNG wire#w4
   // the same network as SCL:
   #_w1 := #MB3_Decoder.Code = #"3033_ROT_RIBALTA";
   "A03_HMI".MB3.Button.A0301.Ribaltatore.Rotazione.Bwd_Minus := #_w1 AND "A0301_Ribaltatore".AreaInterface.Man AND #MB3_Decoder.OperationMinus AND NOT "A0301_Ribaltatore".Ax.DataIn.LS_Minus;
   "A03_HMI".MB3.Button.A0301.Ribaltatore.Rotazione.Fwd_Plus := #_w1 AND "A0301_Ribaltatore".AreaInterface.Man AND #MB3_Decoder.OperationPlus AND NOT "A0301_Ribaltatore".Ax.DataIn.LS_Plus;
   IF #_w1 AND ("A0301_Ribaltatore".COut.Ribaltatore.MinusCheckNext OR "A0301_Ribaltatore".COut.Ribaltatore.PlusCheckNext) THEN
       #MB3_Decoder.OpEnabled := TRUE;
   END_IF;
   IF #_w1 AND (("A0301_Ribaltatore".COut.Ribaltatore.MinusRunning AND NOT "A0301_Ribaltatore".COut.Ribaltatore.MinusLsSwReached) OR ("A0301_Ribaltatore".COut.Ribaltatore.PlusRunning AND NOT "A0301_Ribaltatore".COut.Ribaltatore.PlusLsSwReached)) AND NOT "A0301_Ribaltatore".COut.Ribaltatore.Standstill THEN
       #MB3_Decoder.OpRunning := TRUE;
   END_IF;
   IF #_w1 AND (("A0301_Ribaltatore".COut.Ribaltatore.InPosition AND "A0301_Ribaltatore".COut.Ribaltatore.Standstill) OR "A0301_Ribaltatore".COut.Ribaltatore.MinusLsSwReached OR "A0301_Ribaltatore".COut.Ribaltatore.PlusLsSwReached OR "A0301_Ribaltatore".Ax.DataIn.LS_Minus OR "A0301_Ribaltatore".Ax.DataIn.LS_Plus) THEN
       #MB3_Decoder.OpDone := TRUE;
   END_IF;
END_REGION

